LIN {X 0,Y 340.735,Z 431.04,A -85,B 0,C 180,E1 -14001.773,E2 -14001.773} C_VEL
LIN {X 0,Y 340.725,Z 431.04,A -85,B 0,C 180,E1 -14005.595,E2 -14005.595} C_VEL
LIN {X 0,Y 340.733,Z 431.068,A -85,B 0,C 180,E1 -14009.845,E2 -14009.845} C_VEL
LIN {X 0,Y 343.877,Z 445.891,A -85,B 0,C 180,E1 -14012.952,E2 -14012.952} C_VEL
LIN {X 0,Y 345.184,Z 453.139,A -85,B 0,C 180,E1 -14014.437,E2 -14014.437} C_VEL
LIN {X 0,Y 344.329,Z 467.534,A -85,B 0,C 180,E1 -14017.182,E2 -14017.182} C_VEL
LIN {X 0,Y 343.997,Z 473.692,A -85,B 0,C 180,E1 -14018.325,E2 -14018.325} C_VEL
LIN {X 0,Y 347.393,Z 500.288,A -85,B 0,C 180,E1 -14019.239,E2 -14019.239} C_VEL
LIN {X 0,Y 345.062,Z 584.431,A -85,B 0,C 180,E1 -14021.597,E2 -14021.597} C_VEL
LIN {X 0,Y 344.476,Z 598.904,A -85,B 0,C 180,E1 -14022.256,E2 -14022.256} C_VEL
LIN {X 0,Y 343.764,Z 611.4,A -85,B 0,C 180,E1 -14023.062,E2 -14023.062} C_VEL
LIN {X 0,Y 343.031,Z 623.647,A -85,B 0,C 180,E1 -14024.096,E2 -14024.096} C_VEL
LIN {X 0,Y 342.314,Z 634.938,A -85,B 0,C 180,E1 -14025.308,E2 -14025.308} C_VEL
LIN {X 0,Y 341.516,Z 645.889,A -85,B 0,C 180,E1 -14026.765,E2 -14026.765} C_VEL
LIN {X 0,Y 340.688,Z 655.695,A -85,B 0,C 180,E1 -14028.397,E2 -14028.397} C_VEL
LIN {X 0,Y 340.179,Z 663.039,A -85,B 0,C 180,E1 -14029.886,E2 -14029.886} C_VEL
LIN {X 0,Y 339.671,Z 670.234,A -85,B 0,C 180,E1 -14031.672,E2 -14031.672} C_VEL
LIN {X 0,Y 339.338,Z 676.847,A -85,B 0,C 180,E1 -14033.788,E2 -14033.788} C_VEL
LIN {X 0,Y 339.206,Z 681.571,A -85,B 0,C 180,E1 -14035.841,E2 -14035.841} C_VEL
LIN {X 0,Y 339.05,Z 684.475,A -85,B 0,C 180,E1 -14037.624,E2 -14037.624} C_VEL
LIN {X 0,Y 339.018,Z 685.837,A -85,B 0,C 180,E1 -14038.812,E2 -14038.812} C_VEL
LIN {X 0,Y 339.046,Z 686.75,A -85,B 0,C 180,E1 -14040,E2 -14040} C_VEL
LIN {X 0,Y 339.08,Z 687.194,A -85,B 0,C 180,E1 -14041.188,E2 -14041.188} C_VEL
LIN {X 0,Y 339.136,Z 687.227,A -85,B 0,C 180,E1 -14042.375,E2 -14042.375} C_VEL
LIN {X 0,Y 339.212,Z 686.82,A -85,B 0,C 180,E1 -14043.564,E2 -14043.564} C_VEL
LIN {X 0,Y 339.398,Z 685.947,A -85,B 0,C 180,E1 -14044.751,E2 -14044.751} C_VEL
LIN {X 0,Y 339.705,Z 684.655,A -85,B 0,C 180,E1 -14045.937,E2 -14045.937} C_VEL
LIN {X 0,Y 340.059,Z 681.86,A -85,B 0,C 180,E1 -14047.72,E2 -14047.72} C_VEL
LIN {X 0,Y 340.682,Z 677.987,A -85,B 0,C 180,E1 -14049.499,E2 -14049.499} C_VEL
LIN {X 0,Y 341.571,Z 672.921,A -85,B 0,C 180,E1 -14051.272,E2 -14051.272} C_VEL
LIN {X 0,Y 342.61,Z 666.526,A -85,B 0,C 180,E1 -14053.041,E2 -14053.041} C_VEL
LIN {X 0,Y 344.049,Z 658.543,A -85,B 0,C 180,E1 -14054.794,E2 -14054.794} C_VEL
LIN {X 0,Y 345.341,Z 650.417,A -85,B 0,C 180,E1 -14056.25,E2 -14056.25} C_VEL
LIN {X 0,Y 346.911,Z 640.605,A -85,B 0,C 180,E1 -14057.691,E2 -14057.691} C_VEL
LIN {X 0,Y 348.482,Z 629.771,A -85,B 0,C 180,E1 -14058.978,E2 -14058.978} C_VEL
LIN {X 0,Y 349.949,Z 617.73,A -85,B 0,C 180,E1 -14060.116,E2 -14060.116} C_VEL
LIN {X 0,Y 351.321,Z 605.219,A -85,B 0,C 180,E1 -14061.028,E2 -14061.028} C_VEL
LIN {X 0,Y 352.474,Z 591.942,A -85,B 0,C 180,E1 -14061.761,E2 -14061.761} C_VEL
LIN {X 0,Y 353.611,Z 575.675,A -85,B 0,C 180,E1 -14062.34,E2 -14062.34} C_VEL
LIN {X 0,Y 357.891,Z 509.779,A -85,B 0,C 180,E1 -14064.477,E2 -14064.477} C_VEL
LIN {X 0,Y 358.21,Z 503.514,A -85,B 0,C 180,E1 -14064.704,E2 -14064.704} C_VEL
LIN {X 0,Y 355.972,Z 490.842,A -85,B 0,C 180,E1 -14065.568,E2 -14065.568} C_VEL
LIN {X 0,Y 352.614,Z 476.312,A -85,B 0,C 180,E1 -14066.788,E2 -14066.788} C_VEL
LIN {X 0,Y 353.362,Z 470.45,A -85,B 0,C 180,E1 -14068.018,E2 -14068.018} C_VEL
LIN {X 0,Y 352.553,Z 464.536,A -85,B 0,C 180,E1 -14069.563,E2 -14069.563} C_VEL
LIN {X 0,Y 351.253,Z 458.463,A -85,B 0,C 180,E1 -14071.347,E2 -14071.347} C_VEL
LIN {X 0,Y 349.357,Z 451.655,A -85,B 0,C 180,E1 -14073.608,E2 -14073.608} C_VEL
LIN {X 0,Y 347.334,Z 445.631,A -85,B 0,C 180,E1 -14075.966,E2 -14075.966} C_VEL
LIN {X 0,Y 344.64,Z 439.216,A -85,B 0,C 180,E1 -14079.21,E2 -14079.21} C_VEL
LIN {X 0,Y 342.538,Z 434.998,A -85,B 0,C 180,E1 -14082.385,E2 -14082.385} C_VEL
LIN {X 0,Y 341.197,Z 433.028,A -85,B 0,C 180,E1 -14085.546,E2 -14085.546} C_VEL
LIN {X 0,Y 341.086,Z 432.671,A -85,B 0,C 180,E1 -14087.883,E2 -14087.883} C_VEL
LIN {X 0,Y 341.624,Z 433.725,A -85,B 0,C 180,E1 -14090.376,E2 -14090.376} C_VEL
LIN {X 0,Y 343.462,Z 435.825,A -85,B 0,C 180,E1 -14092.942,E2 -14092.942} C_VEL
LIN {X 0,Y 345.596,Z 439.87,A -85,B 0,C 180,E1 -14095.291,E2 -14095.291} C_VEL
LIN {X 0,Y 346.763,Z 441.759,A -85,B 0,C 180,E1 -14096.198,E2 -14096.198} C_VEL
LIN {X 0,Y 347.63,Z 443.646,A -85,B 0,C 180,E1 -14096.917,E2 -14096.917} C_VEL
LIN {X 0,Y 348.918,Z 451.136,A -85,B 0,C 180,E1 -14098.688,E2 -14098.688} C_VEL
LIN {X 0,Y 351.16,Z 461.414,A -85,B 0,C 180,E1 -14100.754,E2 -14100.754} C_VEL
LIN {X 0,Y 351.367,Z 473.128,A -85,B 0,C 180,E1 -14102.219,E2 -14102.219} C_VEL
LIN {X 0,Y 351.904,Z 484.135,A -85,B 0,C 180,E1 -14103.426,E2 -14103.426} C_VEL
LIN {X 0,Y 354.222,Z 500.627,A -85,B 0,C 180,E1 -14104.573,E2 -14104.573} C_VEL
LIN {X 0,Y 355.496,Z 514.817,A -85,B 0,C 180,E1 -14105.395,E2 -14105.395} C_VEL
LIN {X 0,Y 355.953,Z 529.982,A -85,B 0,C 180,E1 -14106.106,E2 -14106.106} C_VEL
LIN {X 0,Y 351.819,Z 594.042,A -85,B 0,C 180,E1 -14108.234,E2 -14108.234} C_VEL
LIN {X 0,Y 350.644,Z 610.198,A -85,B 0,C 180,E1 -14108.814,E2 -14108.814} C_VEL
LIN {X 0,Y 349.293,Z 624.619,A -85,B 0,C 180,E1 -14109.614,E2 -14109.614} C_VEL
LIN {X 0,Y 347.641,Z 638.466,A -85,B 0,C 180,E1 -14110.668,E2 -14110.668} C_VEL
LIN {X 0,Y 346.154,Z 649.931,A -85,B 0,C 180,E1 -14111.81,E2 -14111.81} C_VEL
LIN {X 0,Y 344.724,Z 660.329,A -85,B 0,C 180,E1 -14113.111,E2 -14113.111} C_VEL
LIN {X 0,Y 343.335,Z 669.83,A -85,B 0,C 180,E1 -14114.567,E2 -14114.567} C_VEL
LIN {X 0,Y 342.004,Z 679.094,A -85,B 0,C 180,E1 -14116.331,E2 -14116.331} C_VEL
LIN {X 0,Y 340.926,Z 686.559,A -85,B 0,C 180,E1 -14118.103,E2 -14118.103} C_VEL
LIN {X 0,Y 340.164,Z 692.472,A -85,B 0,C 180,E1 -14119.885,E2 -14119.885} C_VEL
LIN {X 0,Y 339.571,Z 697.133,A -85,B 0,C 180,E1 -14121.67,E2 -14121.67} C_VEL
LIN {X 0,Y 339.376,Z 699.6,A -85,B 0,C 180,E1 -14122.862,E2 -14122.862} C_VEL
LIN {X 0,Y 339.21,Z 701.57,A -85,B 0,C 180,E1 -14124.054,E2 -14124.054} C_VEL
LIN {X 0,Y 339.155,Z 703.047,A -85,B 0,C 180,E1 -14125.245,E2 -14125.245} C_VEL
LIN {X 0,Y 339.129,Z 704.098,A -85,B 0,C 180,E1 -14126.436,E2 -14126.436} C_VEL
LIN {X 0,Y 339.056,Z 704.68,A -85,B 0,C 180,E1 -14127.624,E2 -14127.624} C_VEL
LIN {X 0,Y 339.14,Z 705.07,A -85,B 0,C 180,E1 -14130,E2 -14130} C_VEL
LIN {X 0,Y 339.076,Z 704.844,A -85,B 0,C 180,E1 -14131.188,E2 -14131.188} C_VEL
LIN {X 0,Y 339.128,Z 703.216,A -85,B 0,C 180,E1 -14133.564,E2 -14133.564} C_VEL
LIN {X 0,Y 339.137,Z 701.78,A -85,B 0,C 180,E1 -14134.755,E2 -14134.755} C_VEL
LIN {X 0,Y 339.239,Z 698.795,A -85,B 0,C 180,E1 -14136.543,E2 -14136.543} C_VEL
LIN {X 0,Y 339.533,Z 694.746,A -85,B 0,C 180,E1 -14138.331,E2 -14138.331} C_VEL
LIN {X 0,Y 340.098,Z 688.503,A -85,B 0,C 180,E1 -14140.417,E2 -14140.417} C_VEL
LIN {X 0,Y 340.817,Z 681.692,A -85,B 0,C 180,E1 -14142.202,E2 -14142.202} C_VEL
LIN {X 0,Y 341.715,Z 674.725,A -85,B 0,C 180,E1 -14143.681,E2 -14143.681} C_VEL
LIN {X 0,Y 342.727,Z 666.304,A -85,B 0,C 180,E1 -14145.156,E2 -14145.156} C_VEL
LIN {X 0,Y 343.843,Z 655.879,A -85,B 0,C 180,E1 -14146.628,E2 -14146.628} C_VEL
LIN {X 0,Y 345.026,Z 645.554,A -85,B 0,C 180,E1 -14147.791,E2 -14147.791} C_VEL
LIN {X 0,Y 346.817,Z 629.693,A -85,B 0,C 180,E1 -14149.226,E2 -14149.226} C_VEL
LIN {X 0,Y 348.632,Z 617.052,A -85,B 0,C 180,E1 -14150.349,E2 -14150.349} C_VEL
LIN {X 0,Y 350.406,Z 603.79,A -85,B 0,C 180,E1 -14151.24,E2 -14151.24} C_VEL
LIN {X 0,Y 351.896,Z 589.543,A -85,B 0,C 180,E1 -14151.953,E2 -14151.953} C_VEL
LIN {X 0,Y 353.266,Z 568.128,A -85,B 0,C 180,E1 -14152.672,E2 -14152.672} C_VEL
LIN {X 0,Y 355.655,Z 527.031,A -85,B 0,C 180,E1 -14154.004,E2 -14154.004} C_VEL
LIN {X 0,Y 354.885,Z 512.697,A -85,B 0,C 180,E1 -14154.691,E2 -14154.691} C_VEL
LIN {X 0,Y 353.058,Z 496.809,A -85,B 0,C 180,E1 -14155.62,E2 -14155.62} C_VEL
LIN {X 0,Y 350.219,Z 481.179,A -85,B 0,C 180,E1 -14156.748,E2 -14156.748} C_VEL
LIN {X 0,Y 347.992,Z 470.293,A -85,B 0,C 180,E1 -14157.678,E2 -14157.678} C_VEL
LIN {X 0,Y 349.181,Z 463.767,A -85,B 0,C 180,E1 -14159.276,E2 -14159.276} C_VEL
LIN {X 0,Y 348.37,Z 458.198,A -85,B 0,C 180,E1 -14160.96,E2 -14160.96} C_VEL
LIN {X 0,Y 346.425,Z 449.389,A -85,B 0,C 180,E1 -14164.025,E2 -14164.025} C_VEL
LIN {X 0,Y 344.561,Z 442.807,A -85,B 0,C 180,E1 -14166.83,E2 -14166.83} C_VEL
LIN {X 0,Y 342.932,Z 437.851,A -85,B 0,C 180,E1 -14169.443,E2 -14169.443} C_VEL
LIN {X 0,Y 341.61,Z 433.699,A -85,B 0,C 180,E1 -14172.214,E2 -14172.214} C_VEL
LIN {X 0,Y 340.674,Z 431.049,A -85,B 0,C 180,E1 -14174.771,E2 -14174.771} C_VEL
LIN {X 0,Y 340.688,Z 431.048,A -85,B 0,C 180,E1 -14178.691,E2 -14178.691} C_VEL
LIN {X 0,Y 340.735,Z 431.041,A -85,B 0,C 180,E1 -14181.773,E2 -14181.773} C_VEL
LIN {X 0,Y 340.725,Z 431.041,A -85,B 0,C 180,E1 -14185.595,E2 -14185.595} C_VEL
LIN {X 0,Y 340.712,Z 431.274,A -85,B 0,C 180,E1 -14187.75,E2 -14187.75} C_VEL
LIN {X 0,Y 341.859,Z 434.768,A -85,B 0,C 180,E1 -14191.111,E2 -14191.111} C_VEL
LIN {X 0,Y 342.024,Z 435.219,A -85,B 0,C 180,E1 -14191.378,E2 -14191.378} C_VEL
LIN {X 0,Y 344.364,Z 438.406,A -85,B 0,C 180,E1 -14192.051,E2 -14192.051} C_VEL
LIN {X 0,Y 346.208,Z 440.911,A -85,B 0,C 180,E1 -14192.546,E2 -14192.546} C_VEL
LIN {X 0,Y 348.676,Z 444.26,A -85,B 0,C 180,E1 -14193.177,E2 -14193.177} C_VEL
LIN {X 0,Y 352.353,Z 449.838,A -85,B 0,C 180,E1 -14194.091,E2 -14194.091} C_VEL
LIN {X 0,Y 357.826,Z 460.119,A -85,B 0,C 180,E1 -14195.413,E2 -14195.413} C_VEL
LIN {X 0,Y 358.798,Z 462.095,A -85,B 0,C 180,E1 -14195.634,E2 -14195.634} C_VEL
LIN {X 0,Y 354.278,Z 529.936,A -85,B 0,C 180,E1 -14197.896,E2 -14197.896} C_VEL
LIN {X 0,Y 353.504,Z 543.651,A -85,B 0,C 180,E1 -14198.497,E2 -14198.497} C_VEL
LIN {X 0,Y 352.576,Z 556.471,A -85,B 0,C 180,E1 -14199.31,E2 -14199.31} C_VEL
LIN {X 0,Y 351.311,Z 568.751,A -85,B 0,C 180,E1 -14200.325,E2 -14200.325} C_VEL
LIN {X 0,Y 349.788,Z 580.474,A -85,B 0,C 180,E1 -14201.551,E2 -14201.551} C_VEL
LIN {X 0,Y 348.228,Z 591.315,A -85,B 0,C 180,E1 -14202.984,E2 -14202.984} C_VEL
LIN {X 0,Y 346.834,Z 600.035,A -85,B 0,C 180,E1 -14204.426,E2 -14204.426} C_VEL
LIN {X 0,Y 345.346,Z 608.53,A -85,B 0,C 180,E1 -14206.165,E2 -14206.165} C_VEL
LIN {X 0,Y 344.008,Z 615.427,A -85,B 0,C 180,E1 -14207.913,E2 -14207.913} C_VEL
LIN {X 0,Y 342.812,Z 621.479,A -85,B 0,C 180,E1 -14209.92,E2 -14209.92} C_VEL
LIN {X 0,Y 341.723,Z 625.627,A -85,B 0,C 180,E1 -14211.723,E2 -14211.723} C_VEL
LIN {X 0,Y 341.324,Z 627.682,A -85,B 0,C 180,E1 -14212.903,E2 -14212.903} C_VEL
LIN {X 0,Y 340.956,Z 629.248,A -85,B 0,C 180,E1 -14214.084,E2 -14214.084} C_VEL
LIN {X 0,Y 340.574,Z 630.401,A -85,B 0,C 180,E1 -14215.265,E2 -14215.265} C_VEL
LIN {X 0,Y 340.191,Z 631.145,A -85,B 0,C 180,E1 -14216.447,E2 -14216.447} C_VEL
LIN {X 0,Y 339.906,Z 631.432,A -85,B 0,C 180,E1 -14217.63,E2 -14217.63} C_VEL
LIN {X 0,Y 339.749,Z 631.264,A -85,B 0,C 180,E1 -14218.815,E2 -14218.815} C_VEL
LIN {X 0,Y 339.693,Z 630.677,A -85,B 0,C 180,E1 -14220,E2 -14220} C_VEL
LIN {X 0,Y 339.712,Z 629.667,A -85,B 0,C 180,E1 -14221.185,E2 -14221.185} C_VEL
LIN {X 0,Y 339.747,Z 628.188,A -85,B 0,C 180,E1 -14222.371,E2 -14222.371} C_VEL
LIN {X 0,Y 340,Z 625.148,A -85,B 0,C 180,E1 -14224.149,E2 -14224.149} C_VEL
LIN {X 0,Y 340.097,Z 621.032,A -85,B 0,C 180,E1 -14225.931,E2 -14225.931} C_VEL
LIN {X 0,Y 340.449,Z 614.758,A -85,B 0,C 180,E1 -14227.993,E2 -14227.993} C_VEL
LIN {X 0,Y 340.865,Z 607.712,A -85,B 0,C 180,E1 -14229.794,E2 -14229.794} C_VEL
LIN {X 0,Y 341.507,Z 599.031,A -85,B 0,C 180,E1 -14231.575,E2 -14231.575} C_VEL
LIN {X 0,Y 342.216,Z 589.175,A -85,B 0,C 180,E1 -14233.207,E2 -14233.207} C_VEL
LIN {X 0,Y 342.969,Z 578.054,A -85,B 0,C 180,E1 -14234.69,E2 -14234.69} C_VEL
LIN {X 0,Y 343.696,Z 566.966,A -85,B 0,C 180,E1 -14235.88,E2 -14235.88} C_VEL
LIN {X 0,Y 344.25,Z 554.855,A -85,B 0,C 180,E1 -14236.913,E2 -14236.913} C_VEL
LIN {X 0,Y 344.841,Z 542.538,A -85,B 0,C 180,E1 -14237.724,E2 -14237.724} C_VEL
LIN {X 0,Y 345.26,Z 529.261,A -85,B 0,C 180,E1 -14238.354,E2 -14238.354} C_VEL
LIN {X 0,Y 345.75,Z 507.069,A -85,B 0,C 180,E1 -14239.017,E2 -14239.017} C_VEL
LIN {X 0,Y 347.211,Z 450.909,A -85,B 0,C 180,E1 -14240.587,E2 -14240.587} C_VEL
LIN {X 0,Y 340.756,Z 431.041,A -85,B 0,C 180,E1 -14241.464,E2 -14241.464} C_VEL
LIN {X 0,Y 340.774,Z 431.037,A -85,B 0,C 180,E1 -14245.664,E2 -14245.664} C_VEL
LIN {X 0,Y 340.731,Z 431.036,A -85,B 0,C 180,E1 -14248.321,E2 -14248.321} C_VEL
LIN {X 0,Y 340.7,Z 431.043,A -85,B 0,C 180,E1 -14251.045,E2 -14251.045} C_VEL
LIN {X 0,Y 340.72,Z 431.031,A -85,B 0,C 180,E1 -14255.279,E2 -14255.279} C_VEL
LIN {X 0,Y 340.712,Z 431.046,A -85,B 0,C 180,E1 -14258.386,E2 -14258.386} C_VEL
LIN {X 0,Y 340.701,Z 431.043,A -85,B 0,C 180,E1 -14262.045,E2 -14262.045} C_VEL
LIN {X 0,Y 340.654,Z 431.038,A -85,B 0,C 180,E1 -14266.227,E2 -14266.227} C_VEL
LIN {X 0,Y 340.69,Z 431.038,A -85,B 0,C 180,E1 -14269.753,E2 -14269.753} C_VEL
LIN {X 0,Y 340.707,Z 431.039,A -85,B 0,C 180,E1 -14273.258,E2 -14273.258} C_VEL
LIN {X 0,Y 340.694,Z 431.043,A -85,B 0,C 180,E1 -14276.153,E2 -14276.153} C_VEL
LIN {X 0,Y 340.73,Z 431.151,A -85,B 0,C 180,E1 -14278.076,E2 -14278.076} C_VEL
LIN {X 0,Y 343.807,Z 443.339,A -85,B 0,C 180,E1 -14280.861,E2 -14280.861} C_VEL
LIN {X 0,Y 346.36,Z 455.442,A -85,B 0,C 180,E1 -14283.487,E2 -14283.487} C_VEL
LIN {X 0,Y 346.577,Z 458.765,A -85,B 0,C 180,E1 -14284.152,E2 -14284.152} C_VEL
LIN {X 0,Y 345.729,Z 472.884,A -85,B 0,C 180,E1 -14286.703,E2 -14286.703} C_VEL
LIN {X 0,Y 350.593,Z 500.147,A -85,B 0,C 180,E1 -14287.657,E2 -14287.657} C_VEL
LIN {X 0,Y 349.247,Z 578.094,A -85,B 0,C 180,E1 -14289.265,E2 -14289.265} C_VEL
LIN {X 0,Y 348.779,Z 591.322,A -85,B 0,C 180,E1 -14289.66,E2 -14289.66} C_VEL
LIN {X 0,Y 347.957,Z 604.505,A -85,B 0,C 180,E1 -14290.303,E2 -14290.303} C_VEL
LIN {X 0,Y 347.044,Z 616.117,A -85,B 0,C 180,E1 -14291.094,E2 -14291.094} C_VEL
LIN {X 0,Y 346.027,Z 627.47,A -85,B 0,C 180,E1 -14292.11,E2 -14292.11} C_VEL
LIN {X 0,Y 344.956,Z 637.518,A -85,B 0,C 180,E1 -14293.249,E2 -14293.249} C_VEL
LIN {X 0,Y 343.897,Z 647.105,A -85,B 0,C 180,E1 -14294.593,E2 -14294.593} C_VEL
LIN {X 0,Y 342.683,Z 655.692,A -85,B 0,C 180,E1 -14296.056,E2 -14296.056} C_VEL
LIN {X 0,Y 341.809,Z 662.776,A -85,B 0,C 180,E1 -14297.532,E2 -14297.532} C_VEL
LIN {X 0,Y 340.928,Z 669.734,A -85,B 0,C 180,E1 -14299.308,E2 -14299.308} C_VEL
LIN {X 0,Y 340.14,Z 675.264,A -85,B 0,C 180,E1 -14301.085,E2 -14301.085} C_VEL
LIN {X 0,Y 339.728,Z 679.599,A -85,B 0,C 180,E1 -14302.87,E2 -14302.87} C_VEL
LIN {X 0,Y 339.498,Z 681.88,A -85,B 0,C 180,E1 -14304.059,E2 -14304.059} C_VEL
LIN {X 0,Y 339.344,Z 683.74,A -85,B 0,C 180,E1 -14305.248,E2 -14305.248} C_VEL
LIN {X 0,Y 339.176,Z 685.162,A -85,B 0,C 180,E1 -14306.436,E2 -14306.436} C_VEL
LIN {X 0,Y 339.057,Z 686.771,A -85,B 0,C 180,E1 -14308.812,E2 -14308.812} C_VEL
LIN {X 0,Y 339.054,Z 687.005,A -85,B 0,C 180,E1 -14310,E2 -14310} C_VEL
LIN {X 0,Y 339.057,Z 686.812,A -85,B 0,C 180,E1 -14311.188,E2 -14311.188} C_VEL
LIN {X 0,Y 339.176,Z 685.257,A -85,B 0,C 180,E1 -14313.564,E2 -14313.564} C_VEL
LIN {X 0,Y 339.341,Z 683.889,A -85,B 0,C 180,E1 -14314.752,E2 -14314.752} C_VEL
LIN {X 0,Y 339.614,Z 680.838,A -85,B 0,C 180,E1 -14316.626,E2 -14316.626} C_VEL
LIN {X 0,Y 339.979,Z 677.11,A -85,B 0,C 180,E1 -14318.32,E2 -14318.32} C_VEL
LIN {X 0,Y 340.594,Z 672.047,A -85,B 0,C 180,E1 -14320.102,E2 -14320.102} C_VEL
LIN {X 0,Y 341.433,Z 665.663,A -85,B 0,C 180,E1 -14321.879,E2 -14321.879} C_VEL
LIN {X 0,Y 342.446,Z 657.73,A -85,B 0,C 180,E1 -14323.651,E2 -14323.651} C_VEL
LIN {X 0,Y 343.587,Z 649.617,A -85,B 0,C 180,E1 -14325.118,E2 -14325.118} C_VEL
LIN {X 0,Y 344.745,Z 639.639,A -85,B 0,C 180,E1 -14326.583,E2 -14326.583} C_VEL
LIN {X 0,Y 345.852,Z 629.069,A -85,B 0,C 180,E1 -14327.828,E2 -14327.828} C_VEL
LIN {X 0,Y 345.787,Z 624.105,A -85,B 0,C 180,E1 -14328.359,E2 -14328.359} C_VEL
LIN {X 0,Y 343.871,Z 615.904,A -85,B 0,C 180,E1 -14329.229,E2 -14329.229} C_VEL
LIN {X 0,Y 341.847,Z 607.372,A -85,B 0,C 180,E1 -14329.998,E2 -14329.998} C_VEL
LIN {X 0,Y 341.6,Z 601.893,A -85,B 0,C 180,E1 -14330.361,E2 -14330.361} C_VEL
LIN {X 0,Y 342.202,Z 589.178,A -85,B 0,C 180,E1 -14330.946,E2 -14330.946} C_VEL
LIN {X 0,Y 342.727,Z 575.953,A -85,B 0,C 180,E1 -14331.306,E2 -14331.306} C_VEL
LIN {X 0,Y 344.073,Z 501.274,A -85,B 0,C 180,E1 -14332.874,E2 -14332.874} C_VEL
LIN {X 0,Y 339.44,Z 475.293,A -85,B 0,C 180,E1 -14333.795,E2 -14333.795} C_VEL
LIN {X 0,Y 339.048,Z 472.783,A -85,B 0,C 180,E1 -14333.933,E2 -14333.933} C_VEL
LIN {X 0,Y 339.88,Z 459.482,A -85,B 0,C 180,E1 -14336.381,E2 -14336.381} C_VEL
LIN {X 0,Y 338.309,Z 450.963,A -85,B 0,C 180,E1 -14338.204,E2 -14338.204} C_VEL
LIN {X 0,Y 335.381,Z 438.328,A -85,B 0,C 180,E1 -14341.086,E2 -14341.086} C_VEL
LIN {X 0,Y 333.648,Z 431.927,A -85,B 0,C 180,E1 -14342.588,E2 -14342.588} C_VEL
LIN {X 0,Y 333.678,Z 431.925,A -85,B 0,C 180,E1 -14346.139,E2 -14346.139} C_VEL
LIN {X 0,Y 333.649,Z 431.924,A -85,B 0,C 180,E1 -14349.192,E2 -14349.192} C_VEL
LIN {X 0,Y 333.635,Z 431.928,A -85,B 0,C 180,E1 -14352.5,E2 -14352.5} C_VEL
LIN {X 0,Y 333.625,Z 431.93,A -85,B 0,C 180,E1 -14355.959,E2 -14355.959} C_VEL
LIN {X 0,Y 333.649,Z 431.92,A -85,B 0,C 180,E1 -14359.315,E2 -14359.315} C_VEL
LIN {X 0,Y 333.667,Z 431.905,A -85,B 0,C 180,E1 -14363.168,E2 -14363.168} C_VEL
LIN {X 0,Y 333.676,Z 431.919,A -85,B 0,C 180,E1 -14365.341,E2 -14365.341} C_VEL
LIN {X 0,Y 333.694,Z 432.008,A -85,B 0,C 180,E1 -14369.594,E2 -14369.594} C_VEL
LIN {X 0,Y 337.063,Z 447.88,A -85,B 0,C 180,E1 -14372.964,E2 -14372.964} C_VEL
LIN {X 0,Y 338.139,Z 453.443,A -85,B 0,C 180,E1 -14374.121,E2 -14374.121} C_VEL
LIN {X 0,Y 337.619,Z 464.884,A -85,B 0,C 180,E1 -14376.337,E2 -14376.337} C_VEL
LIN {X 0,Y 337.043,Z 473.676,A -85,B 0,C 180,E1 -14378.029,E2 -14378.029} C_VEL
LIN {X 0,Y 340.484,Z 500.87,A -85,B 0,C 180,E1 -14378.997,E2 -14378.997} C_VEL
LIN {X 0,Y 338.043,Z 585.238,A -85,B 0,C 180,E1 -14381.437,E2 -14381.437} C_VEL
LIN {X 0,Y 337.444,Z 599.489,A -85,B 0,C 180,E1 -14382.109,E2 -14382.109} C_VEL
LIN {X 0,Y 336.634,Z 612.818,A -85,B 0,C 180,E1 -14383.005,E2 -14383.005} C_VEL
LIN {X 0,Y 335.894,Z 624.819,A -85,B 0,C 180,E1 -14384.061,E2 -14384.061} C_VEL
LIN {X 0,Y 335.164,Z 636.935,A -85,B 0,C 180,E1 -14385.426,E2 -14385.426} C_VEL
LIN {X 0,Y 334.485,Z 645.726,A -85,B 0,C 180,E1 -14386.637,E2 -14386.637} C_VEL
LIN {X 0,Y 333.691,Z 654.815,A -85,B 0,C 180,E1 -14388.15,E2 -14388.15} C_VEL
LIN {X 0,Y 333.039,Z 663.705,A -85,B 0,C 180,E1 -14389.974,E2 -14389.974} C_VEL
LIN {X 0,Y 332.563,Z 670.799,A -85,B 0,C 180,E1 -14391.799,E2 -14391.799} C_VEL
LIN {X 0,Y 332.221,Z 677.252,A -85,B 0,C 180,E1 -14393.928,E2 -14393.928} C_VEL
LIN {X 0,Y 332.122,Z 681.407,A -85,B 0,C 180,E1 -14395.753,E2 -14395.753} C_VEL
LIN {X 0,Y 331.967,Z 684.423,A -85,B 0,C 180,E1 -14397.573,E2 -14397.573} C_VEL
LIN {X 0,Y 331.924,Z 685.841,A -85,B 0,C 180,E1 -14398.787,E2 -14398.787} C_VEL
LIN {X 0,Y 331.949,Z 686.845,A -85,B 0,C 180,E1 -14400,E2 -14400} C_VEL
LIN {X 0,Y 331.985,Z 687.375,A -85,B 0,C 180,E1 -14401.213,E2 -14401.213} C_VEL
LIN {X 0,Y 332.049,Z 687.466,A -85,B 0,C 180,E1 -14402.426,E2 -14402.426} C_VEL
LIN {X 0,Y 332.142,Z 687.143,A -85,B 0,C 180,E1 -14403.639,E2 -14403.639} C_VEL
LIN {X 0,Y 332.351,Z 686.343,A -85,B 0,C 180,E1 -14404.852,E2 -14404.852} C_VEL
LIN {X 0,Y 332.798,Z 683.878,A -85,B 0,C 180,E1 -14407,E2 -14407} C_VEL
LIN {X 0,Y 333.468,Z 680.103,A -85,B 0,C 180,E1 -14409.095,E2 -14409.095} C_VEL
LIN {X 0,Y 334.351,Z 675.57,A -85,B 0,C 180,E1 -14410.905,E2 -14410.905} C_VEL
LIN {X 0,Y 335.557,Z 668.694,A -85,B 0,C 180,E1 -14413.012,E2 -14413.012} C_VEL
LIN {X 0,Y 337.007,Z 661.231,A -85,B 0,C 180,E1 -14414.801,E2 -14414.801} C_VEL
LIN {X 0,Y 338.369,Z 653.636,A -85,B 0,C 180,E1 -14416.284,E2 -14416.284} C_VEL
LIN {X 0,Y 340.028,Z 644.063,A -85,B 0,C 180,E1 -14417.813,E2 -14417.813} C_VEL
LIN {X 0,Y 341.741,Z 633.196,A -85,B 0,C 180,E1 -14419.211,E2 -14419.211} C_VEL
LIN {X 0,Y 343.333,Z 622.142,A -85,B 0,C 180,E1 -14420.364,E2 -14420.364} C_VEL
LIN {X 0,Y 344.862,Z 609.89,A -85,B 0,C 180,E1 -14421.363,E2 -14421.363} C_VEL
LIN {X 0,Y 346.124,Z 597.493,A -85,B 0,C 180,E1 -14422.142,E2 -14422.142} C_VEL
LIN {X 0,Y 347.316,Z 583.091,A -85,B 0,C 180,E1 -14422.768,E2 -14422.768} C_VEL
LIN {X 0,Y 352.794,Z 505.642,A -85,B 0,C 180,E1 -14425.363,E2 -14425.363} C_VEL
LIN {X 0,Y 350.797,Z 493.497,A -85,B 0,C 180,E1 -14426.234,E2 -14426.234} C_VEL
LIN {X 0,Y 347.674,Z 479.394,A -85,B 0,C 180,E1 -14427.463,E2 -14427.463} C_VEL
LIN {X 0,Y 347.038,Z 476.536,A -85,B 0,C 180,E1 -14427.761,E2 -14427.761} C_VEL
LIN {X 0,Y 347.394,Z 472.968,A -85,B 0,C 180,E1 -14428.548,E2 -14428.548} C_VEL
LIN {X 0,Y 346.216,Z 465.172,A -85,B 0,C 180,E1 -14430.748,E2 -14430.748} C_VEL
LIN {X 0,Y 344.233,Z 457.04,A -85,B 0,C 180,E1 -14433.452,E2 -14433.452} C_VEL
LIN {X 0,Y 342.337,Z 450.942,A -85,B 0,C 180,E1 -14435.884,E2 -14435.884} C_VEL
LIN {X 0,Y 340.436,Z 446.072,A -85,B 0,C 180,E1 -14438.327,E2 -14438.327} C_VEL
LIN {X 0,Y 339.288,Z 443.511,A -85,B 0,C 180,E1 -14439.966,E2 -14439.966} C_VEL
LIN {X 0,Y 338.334,Z 441.303,A -85,B 0,C 180,E1 -14441.661,E2 -14441.661} C_VEL
LIN {X 0,Y 337.451,Z 439.778,A -85,B 0,C 180,E1 -14443.416,E2 -14443.416} C_VEL
LIN {X 0,Y 336.859,Z 438.418,A -85,B 0,C 180,E1 -14446.489,E2 -14446.489} C_VEL
LIN {X 0,Y 337.036,Z 438.632,A -85,B 0,C 180,E1 -14448.65,E2 -14448.65} C_VEL
LIN {X 0,Y 338.159,Z 440.394,A -85,B 0,C 180,E1 -14451.428,E2 -14451.428} C_VEL
LIN {X 0,Y 339.584,Z 442.118,A -85,B 0,C 180,E1 -14453.117,E2 -14453.117} C_VEL
LIN {X 0,Y 342.511,Z 447.257,A -85,B 0,C 180,E1 -14455.942,E2 -14455.942} C_VEL
LIN {X 0,Y 343.44,Z 449.705,A -85,B 0,C 180,E1 -14456.815,E2 -14456.815} C_VEL
LIN {X 0,Y 345.163,Z 460.513,A -85,B 0,C 180,E1 -14459.26,E2 -14459.26} C_VEL
LIN {X 0,Y 346.099,Z 464.668,A -85,B 0,C 180,E1 -14460.087,E2 -14460.087} C_VEL
LIN {X 0,Y 346.221,Z 475.224,A -85,B 0,C 180,E1 -14461.486,E2 -14461.486} C_VEL
LIN {X 0,Y 346.444,Z 483.85,A -85,B 0,C 180,E1 -14462.483,E2 -14462.483} C_VEL
LIN {X 0,Y 348.557,Z 498.928,A -85,B 0,C 180,E1 -14463.618,E2 -14463.618} C_VEL
LIN {X 0,Y 350.054,Z 514.876,A -85,B 0,C 180,E1 -14464.617,E2 -14464.617} C_VEL
LIN {X 0,Y 350.418,Z 530.269,A -85,B 0,C 180,E1 -14465.386,E2 -14465.386} C_VEL
LIN {X 0,Y 344.918,Z 607.297,A -85,B 0,C 180,E1 -14468.052,E2 -14468.052} C_VEL
LIN {X 0,Y 343.681,Z 620.288,A -85,B 0,C 180,E1 -14468.717,E2 -14468.717} C_VEL
LIN {X 0,Y 342.249,Z 632.431,A -85,B 0,C 180,E1 -14469.568,E2 -14469.568} C_VEL
LIN {X 0,Y 340.72,Z 643.64,A -85,B 0,C 180,E1 -14470.573,E2 -14470.573} C_VEL
LIN {X 0,Y 339.037,Z 655.101,A -85,B 0,C 180,E1 -14471.884,E2 -14471.884} C_VEL
LIN {X 0,Y 337.582,Z 664.921,A -85,B 0,C 180,E1 -14473.267,E2 -14473.267} C_VEL
LIN {X 0,Y 336.046,Z 674.042,A -85,B 0,C 180,E1 -14474.845,E2 -14474.845} C_VEL
LIN {X 0,Y 334.686,Z 682.385,A -85,B 0,C 180,E1 -14476.645,E2 -14476.645} C_VEL
LIN {X 0,Y 333.669,Z 689.148,A -85,B 0,C 180,E1 -14478.457,E2 -14478.457} C_VEL
LIN {X 0,Y 332.939,Z 694.48,A -85,B 0,C 180,E1 -14480.278,E2 -14480.278} C_VEL
LIN {X 0,Y 332.407,Z 698.594,A -85,B 0,C 180,E1 -14482.101,E2 -14482.101} C_VEL
LIN {X 0,Y 332.12,Z 701.729,A -85,B 0,C 180,E1 -14484.027,E2 -14484.027} C_VEL
LIN {X 0,Y 332.059,Z 703.026,A -85,B 0,C 180,E1 -14485.144,E2 -14485.144} C_VEL
LIN {X 0,Y 332.053,Z 704.01,A -85,B 0,C 180,E1 -14486.359,E2 -14486.359} C_VEL
LIN {X 0,Y 331.991,Z 704.67,A -85,B 0,C 180,E1 -14488.787,E2 -14488.787} C_VEL
LIN {X 0,Y 332.042,Z 704.881,A -85,B 0,C 180,E1 -14490,E2 -14490} C_VEL
LIN {X 0,Y 331.979,Z 704.655,A -85,B 0,C 180,E1 -14491.213,E2 -14491.213} C_VEL
LIN {X 0,Y 332.051,Z 703.027,A -85,B 0,C 180,E1 -14493.641,E2 -14493.641} C_VEL
LIN {X 0,Y 332.076,Z 699.997,A -85,B 0,C 180,E1 -14495.9,E2 -14495.9} C_VEL
LIN {X 0,Y 332.365,Z 696.009,A -85,B 0,C 180,E1 -14497.9,E2 -14497.9} C_VEL
LIN {X 0,Y 332.788,Z 691.191,A -85,B 0,C 180,E1 -14499.727,E2 -14499.727} C_VEL
LIN {X 0,Y 333.402,Z 685.094,A -85,B 0,C 180,E1 -14501.552,E2 -14501.552} C_VEL
LIN {X 0,Y 334.409,Z 677.497,A -85,B 0,C 180,E1 -14503.366,E2 -14503.366} C_VEL
LIN {X 0,Y 335.584,Z 668.106,A -85,B 0,C 180,E1 -14505.141,E2 -14505.141} C_VEL
LIN {X 0,Y 336.719,Z 658.216,A -85,B 0,C 180,E1 -14506.647,E2 -14506.647} C_VEL
LIN {X 0,Y 337.916,Z 648.2,A -85,B 0,C 180,E1 -14507.865,E2 -14507.865} C_VEL
LIN {X 0,Y 339.495,Z 634.856,A -85,B 0,C 180,E1 -14509.186,E2 -14509.186} C_VEL
LIN {X 0,Y 341.59,Z 622.078,A -85,B 0,C 180,E1 -14510.473,E2 -14510.473} C_VEL
LIN {X 0,Y 343.197,Z 611.58,A -85,B 0,C 180,E1 -14511.314,E2 -14511.314} C_VEL
LIN {X 0,Y 344.907,Z 598.324,A -85,B 0,C 180,E1 -14512.146,E2 -14512.146} C_VEL
LIN {X 0,Y 346.36,Z 584.169,A -85,B 0,C 180,E1 -14512.795,E2 -14512.795} C_VEL
LIN {X 0,Y 349.945,Z 527.866,A -85,B 0,C 180,E1 -14514.679,E2 -14514.679} C_VEL
LIN {X 0,Y 349.302,Z 514.056,A -85,B 0,C 180,E1 -14515.369,E2 -14515.369} C_VEL
LIN {X 0,Y 347.643,Z 498.628,A -85,B 0,C 180,E1 -14516.313,E2 -14516.313} C_VEL
LIN {X 0,Y 344.996,Z 483.241,A -85,B 0,C 180,E1 -14517.477,E2 -14517.477} C_VEL
LIN {X 0,Y 342.462,Z 471.523,A -85,B 0,C 180,E1 -14518.524,E2 -14518.524} C_VEL
LIN {X 0,Y 342.078,Z 468.976,A -85,B 0,C 180,E1 -14518.776,E2 -14518.776} C_VEL
LIN {X 0,Y 342.589,Z 466.145,A -85,B 0,C 180,E1 -14519.495,E2 -14519.495} C_VEL
LIN {X 0,Y 341.825,Z 460.54,A -85,B 0,C 180,E1 -14521.25,E2 -14521.25} C_VEL
LIN {X 0,Y 340.044,Z 452.324,A -85,B 0,C 180,E1 -14524.237,E2 -14524.237} C_VEL
LIN {X 0,Y 338.776,Z 447.432,A -85,B 0,C 180,E1 -14526.331,E2 -14526.331} C_VEL
LIN {X 0,Y 336.867,Z 441.494,A -85,B 0,C 180,E1 -14529.473,E2 -14529.473} C_VEL
LIN {X 0,Y 335.625,Z 437.668,A -85,B 0,C 180,E1 -14532.074,E2 -14532.074} C_VEL
LIN {X 0,Y 334.72,Z 435.126,A -85,B 0,C 180,E1 -14534.448,E2 -14534.448} C_VEL
LIN {X 0,Y 333.851,Z 432.972,A -85,B 0,C 180,E1 -14537.651,E2 -14537.651} C_VEL
LIN {X 0,Y 333.722,Z 432.341,A -85,B 0,C 180,E1 -14539.301,E2 -14539.301} C_VEL
LIN {X 0,Y 333.711,Z 432.21,A -85,B 0,C 180,E1 -14542.357,E2 -14542.357} C_VEL
LIN {X 0,Y 333.998,Z 433.297,A -85,B 0,C 180,E1 -14545.38,E2 -14545.38} C_VEL
LIN {X 0,Y 334.475,Z 434.408,A -85,B 0,C 180,E1 -14547.191,E2 -14547.191} C_VEL
LIN {X 0,Y 335.346,Z 437.025,A -85,B 0,C 180,E1 -14549.955,E2 -14549.955} C_VEL
LIN {X 0,Y 337.861,Z 440.383,A -85,B 0,C 180,E1 -14550.787,E2 -14550.787} C_VEL
LIN {X 0,Y 342.02,Z 445.734,A -85,B 0,C 180,E1 -14551.999,E2 -14551.999} C_VEL
LIN {X 0,Y 345.118,Z 450.159,A -85,B 0,C 180,E1 -14552.847,E2 -14552.847} C_VEL
LIN {X 0,Y 348.42,Z 455.366,A -85,B 0,C 180,E1 -14553.72,E2 -14553.72} C_VEL
LIN {X 0,Y 353.244,Z 464.773,A -85,B 0,C 180,E1 -14554.953,E2 -14554.953} C_VEL
LIN {X 0,Y 349.427,Z 515.747,A -85,B 0,C 180,E1 -14556.712,E2 -14556.712} C_VEL
LIN {X 0,Y 348.171,Z 537.01,A -85,B 0,C 180,E1 -14557.487,E2 -14557.487} C_VEL
LIN {X 0,Y 347.286,Z 549.756,A -85,B 0,C 180,E1 -14558.17,E2 -14558.17} C_VEL
LIN {X 0,Y 346.177,Z 562.042,A -85,B 0,C 180,E1 -14559.049,E2 -14559.049} C_VEL
LIN {X 0,Y 344.733,Z 573.959,A -85,B 0,C 180,E1 -14560.144,E2 -14560.144} C_VEL
LIN {X 0,Y 343.254,Z 584.327,A -85,B 0,C 180,E1 -14561.342,E2 -14561.342} C_VEL
LIN {X 0,Y 341.728,Z 593.517,A -85,B 0,C 180,E1 -14562.65,E2 -14562.65} C_VEL
LIN {X 0,Y 340.009,Z 603.567,A -85,B 0,C 180,E1 -14564.412,E2 -14564.412} C_VEL
LIN {X 0,Y 338.415,Z 611.534,A -85,B 0,C 180,E1 -14566.183,E2 -14566.183} C_VEL
LIN {X 0,Y 337.005,Z 617.916,A -85,B 0,C 180,E1 -14567.963,E2 -14567.963} C_VEL
LIN {X 0,Y 336.006,Z 622.616,A -85,B 0,C 180,E1 -14569.627,E2 -14569.627} C_VEL
LIN {X 0,Y 334.811,Z 626.859,A -85,B 0,C 180,E1 -14571.551,E2 -14571.551} C_VEL
LIN {X 0,Y 334.367,Z 628.813,A -85,B 0,C 180,E1 -14572.755,E2 -14572.755} C_VEL
LIN {X 0,Y 333.97,Z 630.296,A -85,B 0,C 180,E1 -14573.96,E2 -14573.96} C_VEL
LIN {X 0,Y 333.565,Z 631.371,A -85,B 0,C 180,E1 -14575.166,E2 -14575.166} C_VEL
LIN {X 0,Y 333.166,Z 632.023,A -85,B 0,C 180,E1 -14576.372,E2 -14576.372} C_VEL
LIN {X 0,Y 332.87,Z 632.205,A -85,B 0,C 180,E1 -14577.58,E2 -14577.58} C_VEL
LIN {X 0,Y 332.706,Z 631.971,A -85,B 0,C 180,E1 -14578.79,E2 -14578.79} C_VEL
LIN {X 0,Y 332.647,Z 631.319,A -85,B 0,C 180,E1 -14580,E2 -14580} C_VEL
LIN {X 0,Y 332.636,Z 630.2,A -85,B 0,C 180,E1 -14581.211,E2 -14581.211} C_VEL
LIN {X 0,Y 332.685,Z 628.647,A -85,B 0,C 180,E1 -14582.422,E2 -14582.422} C_VEL
LIN {X 0,Y 332.948,Z 625.469,A -85,B 0,C 180,E1 -14584.237,E2 -14584.237} C_VEL
LIN {X 0,Y 333.047,Z 621.203,A -85,B 0,C 180,E1 -14586.057,E2 -14586.057} C_VEL
LIN {X 0,Y 333.377,Z 615.044,A -85,B 0,C 180,E1 -14588.075,E2 -14588.075} C_VEL
LIN {X 0,Y 333.835,Z 607.5,A -85,B 0,C 180,E1 -14590.002,E2 -14590.002} C_VEL
LIN {X 0,Y 334.508,Z 598.636,A -85,B 0,C 180,E1 -14591.821,E2 -14591.821} C_VEL
LIN {X 0,Y 335.212,Z 588.486,A -85,B 0,C 180,E1 -14593.488,E2 -14593.488} C_VEL
LIN {X 0,Y 335.947,Z 578.325,A -85,B 0,C 180,E1 -14594.849,E2 -14594.849} C_VEL
LIN {X 0,Y 336.704,Z 567.061,A -85,B 0,C 180,E1 -14596.067,E2 -14596.067} C_VEL
LIN {X 0,Y 337.273,Z 554.869,A -85,B 0,C 180,E1 -14597.118,E2 -14597.118} C_VEL
LIN {X 0,Y 337.883,Z 542.352,A -85,B 0,C 180,E1 -14597.945,E2 -14597.945} C_VEL
LIN {X 0,Y 338.334,Z 527.739,A -85,B 0,C 180,E1 -14598.625,E2 -14598.625} C_VEL
LIN {X 0,Y 340.274,Z 452.148,A -85,B 0,C 180,E1 -14600.819,E2 -14600.819} C_VEL
LIN {X 0,Y 333.71,Z 431.916,A -85,B 0,C 180,E1 -14601.743,E2 -14601.743} C_VEL
LIN {X 0,Y 333.72,Z 431.915,A -85,B 0,C 180,E1 -14605.101,E2 -14605.101} C_VEL
LIN {X 0,Y 333.719,Z 431.908,A -85,B 0,C 180,E1 -14607.809,E2 -14607.809} C_VEL
LIN {X 0,Y 333.692,Z 431.918,A -85,B 0,C 180,E1 -14610.363,E2 -14610.363} C_VEL
LIN {X 0,Y 333.676,Z 431.901,A -85,B 0,C 180,E1 -14614.659,E2 -14614.659} C_VEL
LIN {X 0,Y 333.654,Z 431.925,A -85,B 0,C 180,E1 -14617.651,E2 -14617.651} C_VEL
LIN {X 0,Y 333.648,Z 431.908,A -85,B 0,C 180,E1 -14620.767,E2 -14620.767} C_VEL
LIN {X 0,Y 333.596,Z 431.932,A -85,B 0,C 180,E1 -14624.251,E2 -14624.251} C_VEL
LIN {X 0,Y 333.644,Z 431.925,A -85,B 0,C 180,E1 -14627.619,E2 -14627.619} C_VEL
LIN {X 0,Y 333.655,Z 431.924,A -85,B 0,C 180,E1 -14631.202,E2 -14631.202} C_VEL
LIN {X 0,Y 333.678,Z 431.917,A -85,B 0,C 180,E1 -14633.861,E2 -14633.861} C_VEL
LIN {X 0,Y 333.672,Z 431.962,A -85,B 0,C 180,E1 -14637.56,E2 -14637.56} C_VEL
LIN {X 0,Y 337.046,Z 445.118,A -85,B 0,C 180,E1 -14640.616,E2 -14640.616} C_VEL
LIN {X 0,Y 339.863,Z 458.936,A -85,B 0,C 180,E1 -14643.637,E2 -14643.637} C_VEL
LIN {X 0,Y 339.017,Z 472.991,A -85,B 0,C 180,E1 -14646.212,E2 -14646.212} C_VEL
LIN {X 0,Y 344.047,Z 501.046,A -85,B 0,C 180,E1 -14647.226,E2 -14647.226} C_VEL
LIN {X 0,Y 342.523,Z 579.802,A -85,B 0,C 180,E1 -14648.878,E2 -14648.878} C_VEL
LIN {X 0,Y 342.01,Z 593.171,A -85,B 0,C 180,E1 -14649.317,E2 -14649.317} C_VEL
LIN {X 0,Y 341.213,Z 605.894,A -85,B 0,C 180,E1 -14649.975,E2 -14649.975} C_VEL
LIN {X 0,Y 340.177,Z 618.119,A -85,B 0,C 180,E1 -14650.854,E2 -14650.854} C_VEL
LIN {X 0,Y 339.129,Z 629.024,A -85,B 0,C 180,E1 -14651.889,E2 -14651.889} C_VEL
LIN {X 0,Y 338.016,Z 639.03,A -85,B 0,C 180,E1 -14653.077,E2 -14653.077} C_VEL
LIN {X 0,Y 337.053,Z 647.29,A -85,B 0,C 180,E1 -14654.272,E2 -14654.272} C_VEL
LIN {X 0,Y 335.803,Z 655.878,A -85,B 0,C 180,E1 -14655.764,E2 -14655.764} C_VEL
LIN {X 0,Y 334.868,Z 662.963,A -85,B 0,C 180,E1 -14657.269,E2 -14657.269} C_VEL
LIN {X 0,Y 333.917,Z 669.923,A -85,B 0,C 180,E1 -14659.081,E2 -14659.081} C_VEL
LIN {X 0,Y 333.122,Z 675.453,A -85,B 0,C 180,E1 -14660.896,E2 -14660.896} C_VEL
LIN {X 0,Y 332.674,Z 679.789,A -85,B 0,C 180,E1 -14662.718,E2 -14662.718} C_VEL
LIN {X 0,Y 332.429,Z 682.07,A -85,B 0,C 180,E1 -14663.932,E2 -14663.932} C_VEL
LIN {X 0,Y 332.267,Z 683.93,A -85,B 0,C 180,E1 -14665.147,E2 -14665.147} C_VEL
LIN {X 0,Y 332.107,Z 685.351,A -85,B 0,C 180,E1 -14666.36,E2 -14666.36} C_VEL
LIN {X 0,Y 331.962,Z 686.961,A -85,B 0,C 180,E1 -14668.787,E2 -14668.787} C_VEL
LIN {X 0,Y 331.957,Z 687.194,A -85,B 0,C 180,E1 -14670,E2 -14670} C_VEL
LIN {X 0,Y 331.962,Z 687.001,A -85,B 0,C 180,E1 -14671.213,E2 -14671.213} C_VEL
LIN {X 0,Y 332.106,Z 685.445,A -85,B 0,C 180,E1 -14673.64,E2 -14673.64} C_VEL
LIN {X 0,Y 332.265,Z 684.077,A -85,B 0,C 180,E1 -14674.853,E2 -14674.853} C_VEL
LIN {X 0,Y 332.524,Z 681.331,A -85,B 0,C 180,E1 -14676.604,E2 -14676.604} C_VEL
LIN {X 0,Y 332.933,Z 677.297,A -85,B 0,C 180,E1 -14678.498,E2 -14678.498} C_VEL
LIN {X 0,Y 333.603,Z 672.232,A -85,B 0,C 180,E1 -14680.316,E2 -14680.316} C_VEL
LIN {X 0,Y 334.486,Z 665.846,A -85,B 0,C 180,E1 -14682.129,E2 -14682.129} C_VEL
LIN {X 0,Y 335.54,Z 657.912,A -85,B 0,C 180,E1 -14683.938,E2 -14683.938} C_VEL
LIN {X 0,Y 336.734,Z 649.796,A -85,B 0,C 180,E1 -14685.433,E2 -14685.433} C_VEL
LIN {X 0,Y 337.834,Z 640.982,A -85,B 0,C 180,E1 -14686.771,E2 -14686.771} C_VEL
LIN {X 0,Y 338.873,Z 631.34,A -85,B 0,C 180,E1 -14687.969,E2 -14687.969} C_VEL
LIN {X 0,Y 340.099,Z 619.277,A -85,B 0,C 180,E1 -14689.151,E2 -14689.151} C_VEL
LIN {X 0,Y 341.235,Z 607.531,A -85,B 0,C 180,E1 -14690.024,E2 -14690.024} C_VEL
LIN {X 0,Y 341.6,Z 601.893,A -85,B 0,C 180,E1 -14690.361,E2 -14690.361} C_VEL
LIN {X 0,Y 341.332,Z 596.308,A -85,B 0,C 180,E1 -14690.686,E2 -14690.686} C_VEL
LIN {X 0,Y 339.063,Z 587.196,A -85,B 0,C 180,E1 -14691.228,E2 -14691.228} C_VEL
LIN {X 0,Y 336.641,Z 577.947,A -85,B 0,C 180,E1 -14691.666,E2 -14691.666} C_VEL
LIN {X 0,Y 336.186,Z 572.153,A -85,B 0,C 180,E1 -14691.828,E2 -14691.828} C_VEL
LIN {X 0,Y 337.513,Z 502.096,A -85,B 0,C 180,E1 -14693.327,E2 -14693.327} C_VEL
LIN {X 0,Y 333.066,Z 476.974,A -85,B 0,C 180,E1 -14694.242,E2 -14694.242} C_VEL
LIN {X 0,Y 332.37,Z 473.145,A -85,B 0,C 180,E1 -14694.405,E2 -14694.405} C_VEL
LIN {X 0,Y 333.128,Z 461.458,A -85,B 0,C 180,E1 -14696.561,E2 -14696.561} C_VEL
LIN {X 0,Y 331.848,Z 454.301,A -85,B 0,C 180,E1 -14698.114,E2 -14698.114} C_VEL
LIN {X 0,Y 329.187,Z 442.46,A -85,B 0,C 180,E1 -14700.823,E2 -14700.823} C_VEL
LIN {X 0,Y 326.603,Z 432.805,A -85,B 0,C 180,E1 -14703.126,E2 -14703.126} C_VEL
LIN {X 0,Y 326.632,Z 432.797,A -85,B 0,C 180,E1 -14707.047,E2 -14707.047} C_VEL
LIN {X 0,Y 326.593,Z 432.796,A -85,B 0,C 180,E1 -14710.209,E2 -14710.209} C_VEL
LIN {X 0,Y 326.578,Z 432.797,A -85,B 0,C 180,E1 -14713.523,E2 -14713.523} C_VEL
LIN {X 0,Y 326.585,Z 432.801,A -85,B 0,C 180,E1 -14717.027,E2 -14717.027} C_VEL
LIN {X 0,Y 326.614,Z 432.805,A -85,B 0,C 180,E1 -14720.773,E2 -14720.773} C_VEL
LIN {X 0,Y 326.614,Z 432.787,A -85,B 0,C 180,E1 -14724.48,E2 -14724.48} C_VEL
LIN {X 0,Y 326.61,Z 432.801,A -85,B 0,C 180,E1 -14727.456,E2 -14727.456} C_VEL
LIN {X 0,Y 326.644,Z 432.834,A -85,B 0,C 180,E1 -14729.319,E2 -14729.319} C_VEL
LIN {X 0,Y 330.037,Z 448.766,A -85,B 0,C 180,E1 -14732.741,E2 -14732.741} C_VEL
LIN {X 0,Y 331.228,Z 455.807,A -85,B 0,C 180,E1 -14734.216,E2 -14734.216} C_VEL
LIN {X 0,Y 330.377,Z 469.131,A -85,B 0,C 180,E1 -14736.825,E2 -14736.825} C_VEL
LIN {X 0,Y 330.103,Z 473.904,A -85,B 0,C 180,E1 -14737.738,E2 -14737.738} C_VEL
LIN {X 0,Y 333.507,Z 501.731,A -85,B 0,C 180,E1 -14738.751,E2 -14738.751} C_VEL
LIN {X 0,Y 331.073,Z 585.1,A -85,B 0,C 180,E1 -14741.232,E2 -14741.232} C_VEL
LIN {X 0,Y 330.464,Z 598.694,A -85,B 0,C 180,E1 -14741.879,E2 -14741.879} C_VEL
LIN {X 0,Y 329.826,Z 610.352,A -85,B 0,C 180,E1 -14742.643,E2 -14742.643} C_VEL
LIN {X 0,Y 329.043,Z 622.812,A -85,B 0,C 180,E1 -14743.72,E2 -14743.72} C_VEL
LIN {X 0,Y 328.321,Z 633.748,A -85,B 0,C 180,E1 -14744.906,E2 -14744.906} C_VEL
LIN {X 0,Y 327.503,Z 644.418,A -85,B 0,C 180,E1 -14746.346,E2 -14746.346} C_VEL
LIN {X 0,Y 326.707,Z 653.809,A -85,B 0,C 180,E1 -14747.893,E2 -14747.893} C_VEL
LIN {X 0,Y 326.028,Z 662.893,A -85,B 0,C 180,E1 -14749.756,E2 -14749.756} C_VEL
LIN {X 0,Y 325.5,Z 670.222,A -85,B 0,C 180,E1 -14751.62,E2 -14751.62} C_VEL
LIN {X 0,Y 325.236,Z 675.156,A -85,B 0,C 180,E1 -14753.174,E2 -14753.174} C_VEL
LIN {X 0,Y 325.05,Z 679.873,A -85,B 0,C 180,E1 -14755.038,E2 -14755.038} C_VEL
LIN {X 0,Y 324.932,Z 683.396,A -85,B 0,C 180,E1 -14756.9,E2 -14756.9} C_VEL
LIN {X 0,Y 324.834,Z 685.845,A -85,B 0,C 180,E1 -14758.76,E2 -14758.76} C_VEL
LIN {X 0,Y 324.855,Z 686.911,A -85,B 0,C 180,E1 -14760,E2 -14760} C_VEL
LIN {X 0,Y 324.893,Z 687.55,A -85,B 0,C 180,E1 -14761.239,E2 -14761.239} C_VEL
LIN {X 0,Y 324.964,Z 687.706,A -85,B 0,C 180,E1 -14762.479,E2 -14762.479} C_VEL
LIN {X 0,Y 325.076,Z 687.446,A -85,B 0,C 180,E1 -14763.719,E2 -14763.719} C_VEL
LIN {X 0,Y 325.307,Z 686.766,A -85,B 0,C 180,E1 -14764.957,E2 -14764.957} C_VEL
LIN {X 0,Y 325.762,Z 684.551,A -85,B 0,C 180,E1 -14767.064,E2 -14767.064} C_VEL
LIN {X 0,Y 326.498,Z 680.778,A -85,B 0,C 180,E1 -14769.291,E2 -14769.291} C_VEL
LIN {X 0,Y 327.436,Z 676.426,A -85,B 0,C 180,E1 -14771.138,E2 -14771.138} C_VEL
LIN {X 0,Y 328.726,Z 669.782,A -85,B 0,C 180,E1 -14773.287,E2 -14773.287} C_VEL
LIN {X 0,Y 330.283,Z 662.521,A -85,B 0,C 180,E1 -14775.11,E2 -14775.11} C_VEL
LIN {X 0,Y 331.696,Z 655.119,A -85,B 0,C 180,E1 -14776.621,E2 -14776.621} C_VEL
LIN {X 0,Y 333.461,Z 645.877,A -85,B 0,C 180,E1 -14778.176,E2 -14778.176} C_VEL
LIN {X 0,Y 335.292,Z 635.509,A -85,B 0,C 180,E1 -14779.595,E2 -14779.595} C_VEL
LIN {X 0,Y 337.17,Z 623.34,A -85,B 0,C 180,E1 -14780.913,E2 -14780.913} C_VEL
LIN {X 0,Y 338.748,Z 611.474,A -85,B 0,C 180,E1 -14781.928,E2 -14781.928} C_VEL
LIN {X 0,Y 340.249,Z 598.419,A -85,B 0,C 180,E1 -14782.786,E2 -14782.786} C_VEL
LIN {X 0,Y 341.513,Z 584.713,A -85,B 0,C 180,E1 -14783.418,E2 -14783.418} C_VEL
LIN {X 0,Y 347.136,Z 511.304,A -85,B 0,C 180,E1 -14785.958,E2 -14785.958} C_VEL
LIN {X 0,Y 347.415,Z 506.402,A -85,B 0,C 180,E1 -14786.153,E2 -14786.153} C_VEL
LIN {X 0,Y 345.458,Z 494.582,A -85,B 0,C 180,E1 -14787.064,E2 -14787.064} C_VEL
LIN {X 0,Y 342.764,Z 481.978,A -85,B 0,C 180,E1 -14788.222,E2 -14788.222} C_VEL
LIN {X 0,Y 341.557,Z 476.98,A -85,B 0,C 180,E1 -14788.757,E2 -14788.757} C_VEL
LIN {X 0,Y 340.772,Z 470.188,A -85,B 0,C 180,E1 -14790.693,E2 -14790.693} C_VEL
LIN {X 0,Y 339.181,Z 462.777,A -85,B 0,C 180,E1 -14793.188,E2 -14793.188} C_VEL
LIN {X 0,Y 337.431,Z 456.56,A -85,B 0,C 180,E1 -14795.679,E2 -14795.679} C_VEL
LIN {X 0,Y 335.726,Z 451.635,A -85,B 0,C 180,E1 -14798.194,E2 -14798.194} C_VEL
LIN {X 0,Y 334.673,Z 449.024,A -85,B 0,C 180,E1 -14799.868,E2 -14799.868} C_VEL
LIN {X 0,Y 333.417,Z 446.087,A -85,B 0,C 180,E1 -14802.459,E2 -14802.459} C_VEL
LIN {X 0,Y 332.83,Z 444.944,A -85,B 0,C 180,E1 -14804.173,E2 -14804.173} C_VEL
LIN {X 0,Y 332.579,Z 444.238,A -85,B 0,C 180,E1 -14805.929,E2 -14805.929} C_VEL
LIN {X 0,Y 332.72,Z 444.175,A -85,B 0,C 180,E1 -14807.672,E2 -14807.672} C_VEL
LIN {X 0,Y 333.151,Z 444.821,A -85,B 0,C 180,E1 -14809.415,E2 -14809.415} C_VEL
LIN {X 0,Y 333.977,Z 446.035,A -85,B 0,C 180,E1 -14811.133,E2 -14811.133} C_VEL
LIN {X 0,Y 335.318,Z 447.624,A -85,B 0,C 180,E1 -14812.793,E2 -14812.793} C_VEL
LIN {X 0,Y 337.881,Z 452.112,A -85,B 0,C 180,E1 -14815.385,E2 -14815.385} C_VEL
LIN {X 0,Y 338.759,Z 453.772,A -85,B 0,C 180,E1 -14816.084,E2 -14816.084} C_VEL
LIN {X 0,Y 339.261,Z 457.021,A -85,B 0,C 180,E1 -14816.978,E2 -14816.978} C_VEL
LIN {X 0,Y 340.879,Z 467.023,A -85,B 0,C 180,E1 -14819.205,E2 -14819.205} C_VEL
LIN {X 0,Y 341.251,Z 469.591,A -85,B 0,C 180,E1 -14819.679,E2 -14819.679} C_VEL
LIN {X 0,Y 341.12,Z 481.489,A -85,B 0,C 180,E1 -14821.237,E2 -14821.237} C_VEL
LIN {X 0,Y 341.397,Z 484.768,A -85,B 0,C 180,E1 -14821.591,E2 -14821.591} C_VEL
LIN {X 0,Y 343.32,Z 499.828,A -85,B 0,C 180,E1 -14822.786,E2 -14822.786} C_VEL
LIN {X 0,Y 344.68,Z 514.904,A -85,B 0,C 180,E1 -14823.787,E2 -14823.787} C_VEL
LIN {X 0,Y 344.969,Z 531.844,A -85,B 0,C 180,E1 -14824.67,E2 -14824.67} C_VEL
LIN {X 0,Y 339.106,Z 607.511,A -85,B 0,C 180,E1 -14827.374,E2 -14827.374} C_VEL
LIN {X 0,Y 337.693,Z 620.69,A -85,B 0,C 180,E1 -14828.08,E2 -14828.08} C_VEL
LIN {X 0,Y 336.037,Z 633.419,A -85,B 0,C 180,E1 -14829.013,E2 -14829.013} C_VEL
LIN {X 0,Y 334.183,Z 645.7,A -85,B 0,C 180,E1 -14830.177,E2 -14830.177} C_VEL
LIN {X 0,Y 332.439,Z 656.765,A -85,B 0,C 180,E1 -14831.512,E2 -14831.512} C_VEL
LIN {X 0,Y 330.782,Z 666.784,A -85,B 0,C 180,E1 -14833.031,E2 -14833.031} C_VEL
LIN {X 0,Y 328.988,Z 676.471,A -85,B 0,C 180,E1 -14834.83,E2 -14834.83} C_VEL
LIN {X 0,Y 327.646,Z 684.276,A -85,B 0,C 180,E1 -14836.668,E2 -14836.668} C_VEL
LIN {X 0,Y 326.734,Z 689.612,A -85,B 0,C 180,E1 -14838.209,E2 -14838.209} C_VEL
LIN {X 0,Y 325.946,Z 694.781,A -85,B 0,C 180,E1 -14840.067,E2 -14840.067} C_VEL
LIN {X 0,Y 325.374,Z 698.776,A -85,B 0,C 180,E1 -14841.929,E2 -14841.929} C_VEL
LIN {X 0,Y 325.037,Z 701.995,A -85,B 0,C 180,E1 -14844.055,E2 -14844.055} C_VEL
LIN {X 0,Y 324.957,Z 703.886,A -85,B 0,C 180,E1 -14846.28,E2 -14846.28} C_VEL
LIN {X 0,Y 324.944,Z 704.692,A -85,B 0,C 180,E1 -14850,E2 -14850} C_VEL
LIN {X 0,Y 324.886,Z 704.466,A -85,B 0,C 180,E1 -14851.24,E2 -14851.24} C_VEL
LIN {X 0,Y 324.894,Z 703.847,A -85,B 0,C 180,E1 -14852.48,E2 -14852.48} C_VEL
LIN {X 0,Y 324.953,Z 702.837,A -85,B 0,C 180,E1 -14853.72,E2 -14853.72} C_VEL
LIN {X 0,Y 325.001,Z 700.054,A -85,B 0,C 180,E1 -14855.884,E2 -14855.884} C_VEL
LIN {X 0,Y 325.292,Z 695.819,A -85,B 0,C 180,E1 -14858.073,E2 -14858.073} C_VEL
LIN {X 0,Y 325.772,Z 691.002,A -85,B 0,C 180,E1 -14859.938,E2 -14859.938} C_VEL
LIN {X 0,Y 326.416,Z 684.905,A -85,B 0,C 180,E1 -14861.803,E2 -14861.803} C_VEL
LIN {X 0,Y 327.486,Z 677.309,A -85,B 0,C 180,E1 -14863.654,E2 -14863.654} C_VEL
LIN {X 0,Y 328.668,Z 668.307,A -85,B 0,C 180,E1 -14865.398,E2 -14865.398} C_VEL
LIN {X 0,Y 329.922,Z 657.817,A -85,B 0,C 180,E1 -14867.032,E2 -14867.032} C_VEL
LIN {X 0,Y 331.33,Z 646.607,A -85,B 0,C 180,E1 -14868.392,E2 -14868.392} C_VEL
LIN {X 0,Y 332.207,Z 639.505,A -85,B 0,C 180,E1 -14869.142,E2 -14869.142} C_VEL
LIN {X 0,Y 334.48,Z 626.675,A -85,B 0,C 180,E1 -14870.606,E2 -14870.606} C_VEL
LIN {X 0,Y 336.68,Z 613.868,A -85,B 0,C 180,E1 -14871.748,E2 -14871.748} C_VEL
LIN {X 0,Y 338.784,Z 599.357,A -85,B 0,C 180,E1 -14872.729,E2 -14872.729} C_VEL
LIN {X 0,Y 340.375,Z 585.277,A -85,B 0,C 180,E1 -14873.42,E2 -14873.42} C_VEL
LIN {X 0,Y 344.385,Z 528.538,A -85,B 0,C 180,E1 -14875.398,E2 -14875.398} C_VEL
LIN {X 0,Y 343.791,Z 514.852,A -85,B 0,C 180,E1 -14876.119,E2 -14876.119} C_VEL
LIN {X 0,Y 342.354,Z 500.733,A -85,B 0,C 180,E1 -14877.029,E2 -14877.029} C_VEL
LIN {X 0,Y 340.209,Z 487.066,A -85,B 0,C 180,E1 -14878.097,E2 -14878.097} C_VEL
LIN {X 0,Y 337.281,Z 472.363,A -85,B 0,C 180,E1 -14879.462,E2 -14879.462} C_VEL
LIN {X 0,Y 336,Z 467.498,A -85,B 0,C 180,E1 -14880.058,E2 -14880.058} C_VEL
LIN {X 0,Y 335.04,Z 461.597,A -85,B 0,C 180,E1 -14882.035,E2 -14882.035} C_VEL
LIN {X 0,Y 333.515,Z 454.591,A -85,B 0,C 180,E1 -14884.731,E2 -14884.731} C_VEL
LIN {X 0,Y 332.118,Z 449.474,A -85,B 0,C 180,E1 -14887.091,E2 -14887.091} C_VEL
LIN {X 0,Y 330.726,Z 444.985,A -85,B 0,C 180,E1 -14889.606,E2 -14889.606} C_VEL
LIN {X 0,Y 329.712,Z 441.873,A -85,B 0,C 180,E1 -14891.751,E2 -14891.751} C_VEL
LIN {X 0,Y 328.473,Z 438.404,A -85,B 0,C 180,E1 -14895.084,E2 -14895.084} C_VEL
LIN {X 0,Y 327.743,Z 436.381,A -85,B 0,C 180,E1 -14898.636,E2 -14898.636} C_VEL
LIN {X 0,Y 327.681,Z 435.9,A -85,B 0,C 180,E1 -14901.539,E2 -14901.539} C_VEL
LIN {X 0,Y 327.824,Z 436.66,A -85,B 0,C 180,E1 -14904.631,E2 -14904.631} C_VEL
LIN {X 0,Y 328.45,Z 438.421,A -85,B 0,C 180,E1 -14907.66,E2 -14907.66} C_VEL
LIN {X 0,Y 328.676,Z 439.096,A -85,B 0,C 180,E1 -14908.304,E2 -14908.304} C_VEL
LIN {X 0,Y 330.938,Z 442.047,A -85,B 0,C 180,E1 -14909.179,E2 -14909.179} C_VEL
LIN {X 0,Y 332.616,Z 443.786,A -85,B 0,C 180,E1 -14909.739,E2 -14909.739} C_VEL
LIN {X 0,Y 336.302,Z 448.599,A -85,B 0,C 180,E1 -14910.96,E2 -14910.96} C_VEL
LIN {X 0,Y 338.855,Z 451.985,A -85,B 0,C 180,E1 -14911.713,E2 -14911.713} C_VEL
LIN {X 0,Y 342.929,Z 458.059,A -85,B 0,C 180,E1 -14912.878,E2 -14912.878} C_VEL
LIN {X 0,Y 346.756,Z 465.286,A -85,B 0,C 180,E1 -14913.952,E2 -14913.952} C_VEL
LIN {X 0,Y 347.962,Z 467.874,A -85,B 0,C 180,E1 -14914.277,E2 -14914.277} C_VEL
LIN {X 0,Y 342.906,Z 531.301,A -85,B 0,C 180,E1 -14916.523,E2 -14916.523} C_VEL
LIN {X 0,Y 341.97,Z 545.444,A -85,B 0,C 180,E1 -14917.175,E2 -14917.175} C_VEL
LIN {X 0,Y 341.009,Z 556.729,A -85,B 0,C 180,E1 -14917.906,E2 -14917.906} C_VEL
LIN {X 0,Y 339.53,Z 569.287,A -85,B 0,C 180,E1 -14918.961,E2 -14918.961} C_VEL
LIN {X 0,Y 337.766,Z 581.411,A -85,B 0,C 180,E1 -14920.257,E2 -14920.257} C_VEL
LIN {X 0,Y 335.929,Z 592.189,A -85,B 0,C 180,E1 -14921.711,E2 -14921.711} C_VEL
LIN {X 0,Y 334.347,Z 601.03,A -85,B 0,C 180,E1 -14923.2,E2 -14923.2} C_VEL
LIN {X 0,Y 332.559,Z 609.598,A -85,B 0,C 180,E1 -14924.996,E2 -14924.996} C_VEL
LIN {X 0,Y 330.991,Z 616.574,A -85,B 0,C 180,E1 -14926.806,E2 -14926.806} C_VEL
LIN {X 0,Y 329.571,Z 622.52,A -85,B 0,C 180,E1 -14928.795,E2 -14928.795} C_VEL
LIN {X 0,Y 328.338,Z 626.939,A -85,B 0,C 180,E1 -14930.762,E2 -14930.762} C_VEL
LIN {X 0,Y 327.413,Z 629.924,A -85,B 0,C 180,E1 -14932.6,E2 -14932.6} C_VEL
LIN {X 0,Y 326.986,Z 631.344,A -85,B 0,C 180,E1 -14933.831,E2 -14933.831} C_VEL
LIN {X 0,Y 326.557,Z 632.346,A -85,B 0,C 180,E1 -14935.062,E2 -14935.062} C_VEL
LIN {X 0,Y 326.143,Z 632.881,A -85,B 0,C 180,E1 -14936.293,E2 -14936.293} C_VEL
LIN {X 0,Y 325.835,Z 632.994,A -85,B 0,C 180,E1 -14937.528,E2 -14937.528} C_VEL
LIN {X 0,Y 325.663,Z 632.683,A -85,B 0,C 180,E1 -14938.763,E2 -14938.763} C_VEL
LIN {X 0,Y 325.584,Z 631.919,A -85,B 0,C 180,E1 -14940,E2 -14940} C_VEL
LIN {X 0,Y 325.564,Z 630.716,A -85,B 0,C 180,E1 -14941.237,E2 -14941.237} C_VEL
LIN {X 0,Y 325.689,Z 628.096,A -85,B 0,C 180,E1 -14943.093,E2 -14943.093} C_VEL
LIN {X 0,Y 325.884,Z 624.421,A -85,B 0,C 180,E1 -14944.949,E2 -14944.949} C_VEL
LIN {X 0,Y 326.067,Z 619.594,A -85,B 0,C 180,E1 -14946.808,E2 -14946.808} C_VEL
LIN {X 0,Y 326.379,Z 613.478,A -85,B 0,C 180,E1 -14948.669,E2 -14948.669} C_VEL
LIN {X 0,Y 326.922,Z 605.828,A -85,B 0,C 180,E1 -14950.529,E2 -14950.529} C_VEL
LIN {X 0,Y 327.635,Z 596.317,A -85,B 0,C 180,E1 -14952.387,E2 -14952.387} C_VEL
LIN {X 0,Y 328.376,Z 586.549,A -85,B 0,C 180,E1 -14953.932,E2 -14953.932} C_VEL
LIN {X 0,Y 329.204,Z 574.415,A -85,B 0,C 180,E1 -14955.477,E2 -14955.477} C_VEL
LIN {X 0,Y 329.928,Z 563.135,A -85,B 0,C 180,E1 -14956.621,E2 -14956.621} C_VEL
LIN {X 0,Y 330.539,Z 549.284,A -85,B 0,C 180,E1 -14957.717,E2 -14957.717} C_VEL
LIN {X 0,Y 331.145,Z 535.96,A -85,B 0,C 180,E1 -14958.483,E2 -14958.483} C_VEL
LIN {X 0,Y 331.482,Z 522.247,A -85,B 0,C 180,E1 -14959.025,E2 -14959.025} C_VEL
LIN {X 0,Y 333.368,Z 453.714,A -85,B 0,C 180,E1 -14961.056,E2 -14961.056} C_VEL
LIN {X 0,Y 326.625,Z 432.796,A -85,B 0,C 180,E1 -14962.028,E2 -14962.028} C_VEL
LIN {X 0,Y 326.692,Z 432.793,A -85,B 0,C 180,E1 -14965.484,E2 -14965.484} C_VEL
LIN {X 0,Y 326.65,Z 432.797,A -85,B 0,C 180,E1 -14969.66,E2 -14969.66} C_VEL
LIN {X 0,Y 326.609,Z 432.775,A -85,B 0,C 180,E1 -14974.019,E2 -14974.019} C_VEL
LIN {X 0,Y 326.63,Z 432.803,A -85,B 0,C 180,E1 -14977.239,E2 -14977.239} C_VEL
LIN {X 0,Y 326.579,Z 432.791,A -85,B 0,C 180,E1 -14981.131,E2 -14981.131} C_VEL
LIN {X 0,Y 326.53,Z 432.804,A -85,B 0,C 180,E1 -14984.743,E2 -14984.743} C_VEL
LIN {X 0,Y 326.578,Z 432.806,A -85,B 0,C 180,E1 -14988.154,E2 -14988.154} C_VEL
LIN {X 0,Y 326.625,Z 432.801,A -85,B 0,C 180,E1 -14991.391,E2 -14991.391} C_VEL
LIN {X 0,Y 326.622,Z 432.801,A -85,B 0,C 180,E1 -14994.851,E2 -14994.851} C_VEL
LIN {X 0,Y 326.637,Z 432.973,A -85,B 0,C 180,E1 -14997.049,E2 -14997.049} C_VEL
LIN {X 0,Y 329.853,Z 445.162,A -85,B 0,C 180,E1 -14999.954,E2 -14999.954} C_VEL
LIN {X 0,Y 332.926,Z 459.624,A -85,B 0,C 180,E1 -15003.179,E2 -15003.179} C_VEL
LIN {X 0,Y 332.949,Z 463.939,A -85,B 0,C 180,E1 -15004.024,E2 -15004.024} C_VEL
LIN {X 0,Y 332.347,Z 473.196,A -85,B 0,C 180,E1 -15005.715,E2 -15005.715} C_VEL
LIN {X 0,Y 337.529,Z 502.133,A -85,B 0,C 180,E1 -15006.784,E2 -15006.784} C_VEL
LIN {X 0,Y 335.934,Z 579.913,A -85,B 0,C 180,E1 -15008.443,E2 -15008.443} C_VEL
LIN {X 0,Y 335.401,Z 593.324,A -85,B 0,C 180,E1 -15008.891,E2 -15008.891} C_VEL
LIN {X 0,Y 334.572,Z 606.061,A -85,B 0,C 180,E1 -15009.56,E2 -15009.56} C_VEL
LIN {X 0,Y 333.477,Z 618.295,A -85,B 0,C 180,E1 -15010.454,E2 -15010.454} C_VEL
LIN {X 0,Y 332.197,Z 630.58,A -85,B 0,C 180,E1 -15011.657,E2 -15011.657} C_VEL
LIN {X 0,Y 331.011,Z 641.487,A -85,B 0,C 180,E1 -15013.031,E2 -15013.031} C_VEL
LIN {X 0,Y 329.693,Z 651.113,A -85,B 0,C 180,E1 -15014.546,E2 -15014.546} C_VEL
LIN {X 0,Y 328.231,Z 660.498,A -85,B 0,C 180,E1 -15016.377,E2 -15016.377} C_VEL
LIN {X 0,Y 327.24,Z 667.944,A -85,B 0,C 180,E1 -15018.227,E2 -15018.227} C_VEL
LIN {X 0,Y 326.363,Z 673.921,A -85,B 0,C 180,E1 -15020.08,E2 -15020.08} C_VEL
LIN {X 0,Y 325.758,Z 678.646,A -85,B 0,C 180,E1 -15021.939,E2 -15021.939} C_VEL
LIN {X 0,Y 325.37,Z 682.259,A -85,B 0,C 180,E1 -15023.8,E2 -15023.8} C_VEL
LIN {X 0,Y 325.194,Z 684.119,A -85,B 0,C 180,E1 -15025.041,E2 -15025.041} C_VEL
LIN {X 0,Y 325.04,Z 685.54,A -85,B 0,C 180,E1 -15026.281,E2 -15026.281} C_VEL
LIN {X 0,Y 324.87,Z 687.15,A -85,B 0,C 180,E1 -15028.76,E2 -15028.76} C_VEL
LIN {X 0,Y 324.863,Z 687.383,A -85,B 0,C 180,E1 -15030,E2 -15030} C_VEL
LIN {X 0,Y 324.87,Z 687.19,A -85,B 0,C 180,E1 -15031.24,E2 -15031.24} C_VEL
LIN {X 0,Y 325.039,Z 685.633,A -85,B 0,C 180,E1 -15033.719,E2 -15033.719} C_VEL
LIN {X 0,Y 325.192,Z 684.265,A -85,B 0,C 180,E1 -15034.959,E2 -15034.959} C_VEL
LIN {X 0,Y 325.449,Z 681.76,A -85,B 0,C 180,E1 -15036.604,E2 -15036.604} C_VEL
LIN {X 0,Y 325.898,Z 677.484,A -85,B 0,C 180,E1 -15038.682,E2 -15038.682} C_VEL
LIN {X 0,Y 326.622,Z 672.418,A -85,B 0,C 180,E1 -15040.539,E2 -15040.539} C_VEL
LIN {X 0,Y 327.547,Z 666.03,A -85,B 0,C 180,E1 -15042.39,E2 -15042.39} C_VEL
LIN {X 0,Y 328.655,Z 658.094,A -85,B 0,C 180,E1 -15044.236,E2 -15044.236} C_VEL
LIN {X 0,Y 329.893,Z 649.976,A -85,B 0,C 180,E1 -15045.761,E2 -15045.761} C_VEL
LIN {X 0,Y 331.062,Z 640.651,A -85,B 0,C 180,E1 -15047.197,E2 -15047.197} C_VEL
LIN {X 0,Y 332.294,Z 630.136,A -85,B 0,C 180,E1 -15048.497,E2 -15048.497} C_VEL
LIN {X 0,Y 333.411,Z 619.442,A -85,B 0,C 180,E1 -15049.55,E2 -15049.55} C_VEL
LIN {X 0,Y 334.573,Z 607.685,A -85,B 0,C 180,E1 -15050.44,E2 -15050.44} C_VEL
LIN {X 0,Y 335.34,Z 594.753,A -85,B 0,C 180,E1 -15051.154,E2 -15051.154} C_VEL
LIN {X 0,Y 335.896,Z 582.303,A -85,B 0,C 180,E1 -15051.6,E2 -15051.6} C_VEL
LIN {X 0,Y 336.186,Z 572.153,A -85,B 0,C 180,E1 -15051.828,E2 -15051.828} C_VEL
LIN {X 0,Y 335.782,Z 566.342,A -85,B 0,C 180,E1 -15051.988,E2 -15051.988} C_VEL
LIN {X 0,Y 330.858,Z 547.653,A -85,B 0,C 180,E1 -15052.766,E2 -15052.766} C_VEL
LIN {X 0,Y 330.329,Z 541.842,A -85,B 0,C 180,E1 -15052.94,E2 -15052.94} C_VEL
LIN {X 0,Y 330.968,Z 502.757,A -85,B 0,C 180,E1 -15053.802,E2 -15053.802} C_VEL
LIN {X 0,Y 326.315,Z 476.598,A -85,B 0,C 180,E1 -15054.787,E2 -15054.787} C_VEL
LIN {X 0,Y 325.702,Z 473.237,A -85,B 0,C 180,E1 -15054.94,E2 -15054.94} C_VEL
LIN {X 0,Y 326.345,Z 462.811,A -85,B 0,C 180,E1 -15056.888,E2 -15056.888} C_VEL
LIN {X 0,Y 324.151,Z 451.482,A -85,B 0,C 180,E1 -15059.408,E2 -15059.408} C_VEL
LIN {X 0,Y 321.355,Z 440.34,A -85,B 0,C 180,E1 -15062.029,E2 -15062.029} C_VEL
LIN {X 0,Y 319.57,Z 433.685,A -85,B 0,C 180,E1 -15063.731,E2 -15063.731} C_VEL
LIN {X 0,Y 319.561,Z 433.683,A -85,B 0,C 180,E1 -15066.428,E2 -15066.428} C_VEL
LIN {X 0,Y 319.56,Z 433.674,A -85,B 0,C 180,E1 -15069.669,E2 -15069.669} C_VEL
LIN {X 0,Y 319.559,Z 433.672,A -85,B 0,C 180,E1 -15073.467,E2 -15073.467} C_VEL
LIN {X 0,Y 319.564,Z 433.675,A -85,B 0,C 180,E1 -15077.018,E2 -15077.018} C_VEL
LIN {X 0,Y 319.549,Z 433.682,A -85,B 0,C 180,E1 -15080.371,E2 -15080.371} C_VEL
LIN {X 0,Y 319.561,Z 433.661,A -85,B 0,C 180,E1 -15083.572,E2 -15083.572} C_VEL
LIN {X 0,Y 319.579,Z 433.679,A -85,B 0,C 180,E1 -15086.686,E2 -15086.686} C_VEL
LIN {X 0,Y 319.609,Z 433.693,A -85,B 0,C 180,E1 -15089.047,E2 -15089.047} C_VEL
LIN {X 0,Y 322.896,Z 449.302,A -85,B 0,C 180,E1 -15092.45,E2 -15092.45} C_VEL
LIN {X 0,Y 324.22,Z 456.414,A -85,B 0,C 180,E1 -15093.963,E2 -15093.963} C_VEL
LIN {X 0,Y 323.525,Z 468.273,A -85,B 0,C 180,E1 -15096.316,E2 -15096.316} C_VEL
LIN {X 0,Y 323.201,Z 474.151,A -85,B 0,C 180,E1 -15097.444,E2 -15097.444} C_VEL
LIN {X 0,Y 326.375,Z 499.597,A -85,B 0,C 180,E1 -15098.393,E2 -15098.393} C_VEL
LIN {X 0,Y 326.549,Z 503.931,A -85,B 0,C 180,E1 -15098.538,E2 -15098.538} C_VEL
LIN {X 0,Y 324.037,Z 585.273,A -85,B 0,C 180,E1 -15101.055,E2 -15101.055} C_VEL
LIN {X 0,Y 323.431,Z 598.765,A -85,B 0,C 180,E1 -15101.716,E2 -15101.716} C_VEL
LIN {X 0,Y 322.688,Z 611.372,A -85,B 0,C 180,E1 -15102.574,E2 -15102.574} C_VEL
LIN {X 0,Y 321.867,Z 624.069,A -85,B 0,C 180,E1 -15103.713,E2 -15103.713} C_VEL
LIN {X 0,Y 321.197,Z 634.879,A -85,B 0,C 180,E1 -15104.94,E2 -15104.94} C_VEL
LIN {X 0,Y 320.3,Z 646.112,A -85,B 0,C 180,E1 -15106.518,E2 -15106.518} C_VEL
LIN {X 0,Y 319.434,Z 656.011,A -85,B 0,C 180,E1 -15108.257,E2 -15108.257} C_VEL
LIN {X 0,Y 318.789,Z 664.764,A -85,B 0,C 180,E1 -15110.162,E2 -15110.162} C_VEL
LIN {X 0,Y 318.338,Z 671.728,A -85,B 0,C 180,E1 -15112.069,E2 -15112.069} C_VEL
LIN {X 0,Y 318.036,Z 677.197,A -85,B 0,C 180,E1 -15113.944,E2 -15113.944} C_VEL
LIN {X 0,Y 317.956,Z 680.914,A -85,B 0,C 180,E1 -15115.563,E2 -15115.563} C_VEL
LIN {X 0,Y 317.809,Z 684.213,A -85,B 0,C 180,E1 -15117.465,E2 -15117.465} C_VEL
LIN {X 0,Y 317.747,Z 685.833,A -85,B 0,C 180,E1 -15118.733,E2 -15118.733} C_VEL
LIN {X 0,Y 317.764,Z 686.959,A -85,B 0,C 180,E1 -15120,E2 -15120} C_VEL
LIN {X 0,Y 317.804,Z 687.672,A -85,B 0,C 180,E1 -15121.267,E2 -15121.267} C_VEL
LIN {X 0,Y 317.883,Z 687.951,A -85,B 0,C 180,E1 -15122.534,E2 -15122.534} C_VEL
LIN {X 0,Y 318.013,Z 687.755,A -85,B 0,C 180,E1 -15123.801,E2 -15123.801} C_VEL
LIN {X 0,Y 318.265,Z 687.145,A -85,B 0,C 180,E1 -15125.067,E2 -15125.067} C_VEL
LIN {X 0,Y 318.729,Z 685.211,A -85,B 0,C 180,E1 -15127.134,E2 -15127.134} C_VEL
LIN {X 0,Y 319.54,Z 681.505,A -85,B 0,C 180,E1 -15129.495,E2 -15129.495} C_VEL
LIN {X 0,Y 320.531,Z 677.306,A -85,B 0,C 180,E1 -15131.381,E2 -15131.381} C_VEL
LIN {X 0,Y 321.65,Z 671.91,A -85,B 0,C 180,E1 -15133.263,E2 -15133.263} C_VEL
LIN {X 0,Y 323.247,Z 665.12,A -85,B 0,C 180,E1 -15135.124,E2 -15135.124} C_VEL
LIN {X 0,Y 325.062,Z 656.723,A -85,B 0,C 180,E1 -15136.97,E2 -15136.97} C_VEL
LIN {X 0,Y 327.036,Z 647.257,A -85,B 0,C 180,E1 -15138.633,E2 -15138.633} C_VEL
LIN {X 0,Y 329.25,Z 635.413,A -85,B 0,C 180,E1 -15140.296,E2 -15140.296} C_VEL
LIN {X 0,Y 331.296,Z 623.332,A -85,B 0,C 180,E1 -15141.629,E2 -15141.629} C_VEL
LIN {X 0,Y 333,Z 611.495,A -85,B 0,C 180,E1 -15142.654,E2 -15142.654} C_VEL
LIN {X 0,Y 334.574,Z 598.396,A -85,B 0,C 180,E1 -15143.523,E2 -15143.523} C_VEL
LIN {X 0,Y 336.076,Z 582.891,A -85,B 0,C 180,E1 -15144.23,E2 -15144.23} C_VEL
LIN {X 0,Y 342.29,Z 508.601,A -85,B 0,C 180,E1 -15146.887,E2 -15146.887} C_VEL
LIN {X 0,Y 340.518,Z 497.148,A -85,B 0,C 180,E1 -15147.81,E2 -15147.81} C_VEL
LIN {X 0,Y 338.05,Z 484.788,A -85,B 0,C 180,E1 -15149.002,E2 -15149.002} C_VEL
LIN {X 0,Y 336.971,Z 480.702,A -85,B 0,C 180,E1 -15149.481,E2 -15149.481} C_VEL
LIN {X 0,Y 335.554,Z 477.183,A -85,B 0,C 180,E1 -15150.07,E2 -15150.07} C_VEL
LIN {X 0,Y 334.595,Z 471.125,A -85,B 0,C 180,E1 -15152.014,E2 -15152.014} C_VEL
LIN {X 0,Y 333.086,Z 464.192,A -85,B 0,C 180,E1 -15154.625,E2 -15154.625} C_VEL
LIN {X 0,Y 331.477,Z 458.542,A -85,B 0,C 180,E1 -15157.274,E2 -15157.274} C_VEL
LIN {X 0,Y 329.978,Z 454.336,A -85,B 0,C 180,E1 -15159.937,E2 -15159.937} C_VEL
LIN {X 0,Y 329.199,Z 452.421,A -85,B 0,C 180,E1 -15161.651,E2 -15161.651} C_VEL
LIN {X 0,Y 328.667,Z 451.059,A -85,B 0,C 180,E1 -15163.361,E2 -15163.361} C_VEL
LIN {X 0,Y 328.375,Z 450.221,A -85,B 0,C 180,E1 -15165.067,E2 -15165.067} C_VEL
LIN {X 0,Y 328.412,Z 449.896,A -85,B 0,C 180,E1 -15166.78,E2 -15166.78} C_VEL
LIN {X 0,Y 328.732,Z 450.2,A -85,B 0,C 180,E1 -15168.49,E2 -15168.49} C_VEL
LIN {X 0,Y 329.437,Z 451.176,A -85,B 0,C 180,E1 -15170.208,E2 -15170.208} C_VEL
LIN {X 0,Y 331.365,Z 453.626,A -85,B 0,C 180,E1 -15172.809,E2 -15172.809} C_VEL
LIN {X 0,Y 333.96,Z 458.156,A -85,B 0,C 180,E1 -15175.375,E2 -15175.375} C_VEL
LIN {X 0,Y 334.622,Z 460.085,A -85,B 0,C 180,E1 -15176.074,E2 -15176.074} C_VEL
LIN {X 0,Y 336,Z 470.312,A -85,B 0,C 180,E1 -15178.472,E2 -15178.472} C_VEL
LIN {X 0,Y 336.4,Z 473.541,A -85,B 0,C 180,E1 -15179.094,E2 -15179.094} C_VEL
LIN {X 0,Y 336.16,Z 483.518,A -85,B 0,C 180,E1 -15180.424,E2 -15180.424} C_VEL
LIN {X 0,Y 337.951,Z 497.287,A -85,B 0,C 180,E1 -15181.641,E2 -15181.641} C_VEL
LIN {X 0,Y 339.325,Z 512.708,A -85,B 0,C 180,E1 -15182.767,E2 -15182.767} C_VEL
LIN {X 0,Y 339.69,Z 523.87,A -85,B 0,C 180,E1 -15183.418,E2 -15183.418} C_VEL
LIN {X 0,Y 339.667,Z 533.167,A -85,B 0,C 180,E1 -15183.902,E2 -15183.902} C_VEL
LIN {X 0,Y 333.422,Z 607.21,A -85,B 0,C 180,E1 -15186.638,E2 -15186.638} C_VEL
LIN {X 0,Y 331.76,Z 621.32,A -85,B 0,C 180,E1 -15187.421,E2 -15187.421} C_VEL
LIN {X 0,Y 330.147,Z 632.994,A -85,B 0,C 180,E1 -15188.292,E2 -15188.292} C_VEL
LIN {X 0,Y 328.18,Z 645.199,A -85,B 0,C 180,E1 -15189.471,E2 -15189.471} C_VEL
LIN {X 0,Y 326.26,Z 656.191,A -85,B 0,C 180,E1 -15190.822,E2 -15190.822} C_VEL
LIN {X 0,Y 324.361,Z 666.692,A -85,B 0,C 180,E1 -15192.432,E2 -15192.432} C_VEL
LIN {X 0,Y 322.5,Z 675.992,A -85,B 0,C 180,E1 -15194.193,E2 -15194.193} C_VEL
LIN {X 0,Y 320.955,Z 683.796,A -85,B 0,C 180,E1 -15196.062,E2 -15196.062} C_VEL
LIN {X 0,Y 319.811,Z 690.134,A -85,B 0,C 180,E1 -15197.95,E2 -15197.95} C_VEL
LIN {X 0,Y 318.961,Z 695.151,A -85,B 0,C 180,E1 -15199.847,E2 -15199.847} C_VEL
LIN {X 0,Y 318.338,Z 698.978,A -85,B 0,C 180,E1 -15201.749,E2 -15201.749} C_VEL
LIN {X 0,Y 317.95,Z 702.192,A -85,B 0,C 180,E1 -15204.091,E2 -15204.091} C_VEL
LIN {X 0,Y 317.863,Z 703.769,A -85,B 0,C 180,E1 -15206.197,E2 -15206.197} C_VEL
LIN {X 0,Y 317.849,Z 704.503,A -85,B 0,C 180,E1 -15210,E2 -15210} C_VEL
LIN {X 0,Y 317.795,Z 704.277,A -85,B 0,C 180,E1 -15211.267,E2 -15211.267} C_VEL
LIN {X 0,Y 317.813,Z 703.658,A -85,B 0,C 180,E1 -15212.535,E2 -15212.535} C_VEL
LIN {X 0,Y 317.859,Z 702.648,A -85,B 0,C 180,E1 -15213.803,E2 -15213.803} C_VEL
LIN {X 0,Y 317.894,Z 700.173,A -85,B 0,C 180,E1 -15215.81,E2 -15215.81} C_VEL
LIN {X 0,Y 318.116,Z 696.984,A -85,B 0,C 180,E1 -15217.617,E2 -15217.617} C_VEL
LIN {X 0,Y 318.549,Z 692.563,A -85,B 0,C 180,E1 -15219.525,E2 -15219.525} C_VEL
LIN {X 0,Y 319.166,Z 686.927,A -85,B 0,C 180,E1 -15221.431,E2 -15221.431} C_VEL
LIN {X 0,Y 320.183,Z 679.834,A -85,B 0,C 180,E1 -15223.325,E2 -15223.325} C_VEL
LIN {X 0,Y 321.367,Z 670.973,A -85,B 0,C 180,E1 -15225.214,E2 -15225.214} C_VEL
LIN {X 0,Y 322.605,Z 661.866,A -85,B 0,C 180,E1 -15226.777,E2 -15226.777} C_VEL
LIN {X 0,Y 323.905,Z 651.727,A -85,B 0,C 180,E1 -15228.174,E2 -15228.174} C_VEL
LIN {X 0,Y 325.157,Z 642.689,A -85,B 0,C 180,E1 -15229.246,E2 -15229.246} C_VEL
LIN {X 0,Y 327.484,Z 630.901,A -85,B 0,C 180,E1 -15230.738,E2 -15230.738} C_VEL
LIN {X 0,Y 329.595,Z 619.446,A -85,B 0,C 180,E1 -15231.91,E2 -15231.91} C_VEL
LIN {X 0,Y 331.918,Z 605.886,A -85,B 0,C 180,E1 -15232.979,E2 -15232.979} C_VEL
LIN {X 0,Y 333.792,Z 593.15,A -85,B 0,C 180,E1 -15233.746,E2 -15233.746} C_VEL
LIN {X 0,Y 335.128,Z 579.984,A -85,B 0,C 180,E1 -15234.344,E2 -15234.344} C_VEL
LIN {X 0,Y 338.929,Z 529.526,A -85,B 0,C 180,E1 -15236.146,E2 -15236.146} C_VEL
LIN {X 0,Y 338.469,Z 516.272,A -85,B 0,C 180,E1 -15236.874,E2 -15236.874} C_VEL
LIN {X 0,Y 337.172,Z 502.417,A -85,B 0,C 180,E1 -15237.811,E2 -15237.811} C_VEL
LIN {X 0,Y 335.241,Z 489.17,A -85,B 0,C 180,E1 -15238.896,E2 -15238.896} C_VEL
LIN {X 0,Y 332.646,Z 475.398,A -85,B 0,C 180,E1 -15240.245,E2 -15240.245} C_VEL
LIN {X 0,Y 331.579,Z 471.745,A -85,B 0,C 180,E1 -15240.714,E2 -15240.714} C_VEL
LIN {X 0,Y 328.825,Z 465.479,A -85,B 0,C 180,E1 -15241.84,E2 -15241.84} C_VEL
LIN {X 0,Y 327.482,Z 458.974,A -85,B 0,C 180,E1 -15244.363,E2 -15244.363} C_VEL
LIN {X 0,Y 325.973,Z 453.023,A -85,B 0,C 180,E1 -15247.134,E2 -15247.134} C_VEL
LIN {X 0,Y 324.577,Z 448.447,A -85,B 0,C 180,E1 -15249.766,E2 -15249.766} C_VEL
LIN {X 0,Y 323.415,Z 444.934,A -85,B 0,C 180,E1 -15252.367,E2 -15252.367} C_VEL
LIN {X 0,Y 322.747,Z 443.056,A -85,B 0,C 180,E1 -15254.172,E2 -15254.172} C_VEL
LIN {X 0,Y 321.888,Z 440.789,A -85,B 0,C 180,E1 -15257.402,E2 -15257.402} C_VEL
LIN {X 0,Y 321.677,Z 439.746,A -85,B 0,C 180,E1 -15260.684,E2 -15260.684} C_VEL
LIN {X 0,Y 321.703,Z 439.751,A -85,B 0,C 180,E1 -15262.288,E2 -15262.288} C_VEL
LIN {X 0,Y 322.05,Z 441.15,A -85,B 0,C 180,E1 -15266.204,E2 -15266.204} C_VEL
LIN {X 0,Y 323.339,Z 443.035,A -85,B 0,C 180,E1 -15266.931,E2 -15266.931} C_VEL
LIN {X 0,Y 326.04,Z 445.709,A -85,B 0,C 180,E1 -15268.047,E2 -15268.047} C_VEL
LIN {X 0,Y 328.944,Z 449.026,A -85,B 0,C 180,E1 -15269.151,E2 -15269.151} C_VEL
LIN {X 0,Y 333.336,Z 454.917,A -85,B 0,C 180,E1 -15270.681,E2 -15270.681} C_VEL
LIN {X 0,Y 337.033,Z 460.145,A -85,B 0,C 180,E1 -15271.83,E2 -15271.83} C_VEL
LIN {X 0,Y 340.789,Z 466.587,A -85,B 0,C 180,E1 -15272.953,E2 -15272.953} C_VEL
LIN {X 0,Y 342.722,Z 470.945,A -85,B 0,C 180,E1 -15273.54,E2 -15273.54} C_VEL
LIN {X 0,Y 337.416,Z 532.467,A -85,B 0,C 180,E1 -15275.791,E2 -15275.791} C_VEL
LIN {X 0,Y 336.439,Z 545.574,A -85,B 0,C 180,E1 -15276.412,E2 -15276.412} C_VEL
LIN {X 0,Y 335.148,Z 559.103,A -85,B 0,C 180,E1 -15277.321,E2 -15277.321} C_VEL
LIN {X 0,Y 333.581,Z 571.352,A -85,B 0,C 180,E1 -15278.387,E2 -15278.387} C_VEL
LIN {X 0,Y 331.934,Z 581.953,A -85,B 0,C 180,E1 -15279.552,E2 -15279.552} C_VEL
LIN {X 0,Y 329.898,Z 592.789,A -85,B 0,C 180,E1 -15281.042,E2 -15281.042} C_VEL
LIN {X 0,Y 328.192,Z 601.663,A -85,B 0,C 180,E1 -15282.554,E2 -15282.554} C_VEL
LIN {X 0,Y 326.248,Z 610.311,A -85,B 0,C 180,E1 -15284.379,E2 -15284.379} C_VEL
LIN {X 0,Y 324.54,Z 617.246,A -85,B 0,C 180,E1 -15286.219,E2 -15286.219} C_VEL
LIN {X 0,Y 322.892,Z 623.517,A -85,B 0,C 180,E1 -15288.368,E2 -15288.368} C_VEL
LIN {X 0,Y 321.452,Z 628.255,A -85,B 0,C 180,E1 -15290.562,E2 -15290.562} C_VEL
LIN {X 0,Y 320.468,Z 631.089,A -85,B 0,C 180,E1 -15292.439,E2 -15292.439} C_VEL
LIN {X 0,Y 320.007,Z 632.416,A -85,B 0,C 180,E1 -15293.696,E2 -15293.696} C_VEL
LIN {X 0,Y 319.55,Z 633.281,A -85,B 0,C 180,E1 -15294.953,E2 -15294.953} C_VEL
LIN {X 0,Y 319.121,Z 633.733,A -85,B 0,C 180,E1 -15296.212,E2 -15296.212} C_VEL
LIN {X 0,Y 318.802,Z 633.773,A -85,B 0,C 180,E1 -15297.473,E2 -15297.473} C_VEL
LIN {X 0,Y 318.621,Z 633.362,A -85,B 0,C 180,E1 -15298.736,E2 -15298.736} C_VEL
LIN {X 0,Y 318.509,Z 632.498,A -85,B 0,C 180,E1 -15300,E2 -15300} C_VEL
LIN {X 0,Y 318.493,Z 631.215,A -85,B 0,C 180,E1 -15301.264,E2 -15301.264} C_VEL
LIN {X 0,Y 318.632,Z 628.449,A -85,B 0,C 180,E1 -15303.161,E2 -15303.161} C_VEL
LIN {X 0,Y 318.806,Z 624.631,A -85,B 0,C 180,E1 -15305.059,E2 -15305.059} C_VEL
LIN {X 0,Y 319.03,Z 618.858,A -85,B 0,C 180,E1 -15307.223,E2 -15307.223} C_VEL
LIN {X 0,Y 319.415,Z 612.127,A -85,B 0,C 180,E1 -15309.179,E2 -15309.179} C_VEL
LIN {X 0,Y 320.054,Z 603.989,A -85,B 0,C 180,E1 -15311.078,E2 -15311.078} C_VEL
LIN {X 0,Y 320.625,Z 595.659,A -85,B 0,C 180,E1 -15312.662,E2 -15312.662} C_VEL
LIN {X 0,Y 321.5,Z 584.421,A -85,B 0,C 180,E1 -15314.398,E2 -15314.398} C_VEL
LIN {X 0,Y 322.301,Z 572.943,A -85,B 0,C 180,E1 -15315.817,E2 -15315.817} C_VEL
LIN {X 0,Y 323.062,Z 560.1,A -85,B 0,C 180,E1 -15317.078,E2 -15317.078} C_VEL
LIN {X 0,Y 323.641,Z 547.511,A -85,B 0,C 180,E1 -15318.026,E2 -15318.026} C_VEL
LIN {X 0,Y 324.226,Z 533.31,A -85,B 0,C 180,E1 -15318.81,E2 -15318.81} C_VEL
LIN {X 0,Y 324.598,Z 516.462,A -85,B 0,C 180,E1 -15319.403,E2 -15319.403} C_VEL
LIN {X 0,Y 326.507,Z 455.246,A -85,B 0,C 180,E1 -15321.28,E2 -15321.28} C_VEL
LIN {X 0,Y 319.589,Z 433.672,A -85,B 0,C 180,E1 -15322.294,E2 -15322.294} C_VEL
LIN {X 0,Y 319.62,Z 433.67,A -85,B 0,C 180,E1 -15326.09,E2 -15326.09} C_VEL
LIN {X 0,Y 319.582,Z 433.673,A -85,B 0,C 180,E1 -15328.935,E2 -15328.935} C_VEL
LIN {X 0,Y 319.533,Z 433.672,A -85,B 0,C 180,E1 -15331.862,E2 -15331.862} C_VEL
LIN {X 0,Y 319.582,Z 433.666,A -85,B 0,C 180,E1 -15335.543,E2 -15335.543} C_VEL
LIN {X 0,Y 319.575,Z 433.679,A -85,B 0,C 180,E1 -15338.008,E2 -15338.008} C_VEL
LIN {X 0,Y 319.528,Z 433.674,A -85,B 0,C 180,E1 -15341.597,E2 -15341.597} C_VEL
LIN {X 0,Y 319.49,Z 433.675,A -85,B 0,C 180,E1 -15345.257,E2 -15345.257} C_VEL
LIN {X 0,Y 319.53,Z 433.68,A -85,B 0,C 180,E1 -15348.712,E2 -15348.712} C_VEL
LIN {X 0,Y 319.579,Z 433.675,A -85,B 0,C 180,E1 -15352.344,E2 -15352.344} C_VEL
LIN {X 0,Y 319.569,Z 433.674,A -85,B 0,C 180,E1 -15356.269,E2 -15356.269} C_VEL
LIN {X 0,Y 319.586,Z 433.759,A -85,B 0,C 180,E1 -15356.479,E2 -15356.479} C_VEL
LIN {X 0,Y 323.437,Z 448.445,A -85,B 0,C 180,E1 -15360.015,E2 -15360.015} C_VEL
LIN {X 0,Y 326.314,Z 462.259,A -85,B 0,C 180,E1 -15363.109,E2 -15363.109} C_VEL
LIN {X 0,Y 325.683,Z 473.289,A -85,B 0,C 180,E1 -15365.183,E2 -15365.183} C_VEL
LIN {X 0,Y 330.444,Z 499.684,A -85,B 0,C 180,E1 -15366.196,E2 -15366.196} C_VEL
LIN {X 0,Y 331.048,Z 503.636,A -85,B 0,C 180,E1 -15366.335,E2 -15366.335} C_VEL
LIN {X 0,Y 329.359,Z 580.024,A -85,B 0,C 180,E1 -15367.991,E2 -15367.991} C_VEL
LIN {X 0,Y 328.84,Z 592.637,A -85,B 0,C 180,E1 -15368.408,E2 -15368.408} C_VEL
LIN {X 0,Y 328.036,Z 605.004,A -85,B 0,C 180,E1 -15369.052,E2 -15369.052} C_VEL
LIN {X 0,Y 327.015,Z 616.639,A -85,B 0,C 180,E1 -15369.888,E2 -15369.888} C_VEL
LIN {X 0,Y 325.83,Z 628.009,A -85,B 0,C 180,E1 -15370.959,E2 -15370.959} C_VEL
LIN {X 0,Y 324.592,Z 638.26,A -85,B 0,C 180,E1 -15372.192,E2 -15372.192} C_VEL
LIN {X 0,Y 323.417,Z 647.66,A -85,B 0,C 180,E1 -15373.591,E2 -15373.591} C_VEL
LIN {X 0,Y 322.077,Z 656.251,A -85,B 0,C 180,E1 -15375.144,E2 -15375.144} C_VEL
LIN {X 0,Y 320.971,Z 663.34,A -85,B 0,C 180,E1 -15376.708,E2 -15376.708} C_VEL
LIN {X 0,Y 319.984,Z 670.3,A -85,B 0,C 180,E1 -15378.599,E2 -15378.599} C_VEL
LIN {X 0,Y 319.101,Z 675.831,A -85,B 0,C 180,E1 -15380.492,E2 -15380.492} C_VEL
LIN {X 0,Y 318.58,Z 680.167,A -85,B 0,C 180,E1 -15382.394,E2 -15382.394} C_VEL
LIN {X 0,Y 318.316,Z 682.449,A -85,B 0,C 180,E1 -15383.662,E2 -15383.662} C_VEL
LIN {X 0,Y 318.124,Z 684.309,A -85,B 0,C 180,E1 -15384.93,E2 -15384.93} C_VEL
LIN {X 0,Y 317.974,Z 685.729,A -85,B 0,C 180,E1 -15386.198,E2 -15386.198} C_VEL
LIN {X 0,Y 317.781,Z 687.339,A -85,B 0,C 180,E1 -15388.733,E2 -15388.733} C_VEL
LIN {X 0,Y 317.771,Z 687.572,A -85,B 0,C 180,E1 -15390,E2 -15390} C_VEL
LIN {X 0,Y 317.781,Z 687.379,A -85,B 0,C 180,E1 -15391.267,E2 -15391.267} C_VEL
LIN {X 0,Y 317.973,Z 685.821,A -85,B 0,C 180,E1 -15393.802,E2 -15393.802} C_VEL
LIN {X 0,Y 318.122,Z 684.453,A -85,B 0,C 180,E1 -15395.07,E2 -15395.07} C_VEL
LIN {X 0,Y 318.342,Z 682.27,A -85,B 0,C 180,E1 -15396.554,E2 -15396.554} C_VEL
LIN {X 0,Y 318.886,Z 677.67,A -85,B 0,C 180,E1 -15398.875,E2 -15398.875} C_VEL
LIN {X 0,Y 319.634,Z 672.603,A -85,B 0,C 180,E1 -15400.772,E2 -15400.772} C_VEL
LIN {X 0,Y 320.596,Z 666.215,A -85,B 0,C 180,E1 -15402.663,E2 -15402.663} C_VEL
LIN {X 0,Y 321.787,Z 658.275,A -85,B 0,C 180,E1 -15404.547,E2 -15404.547} C_VEL
LIN {X 0,Y 323.069,Z 650.155,A -85,B 0,C 180,E1 -15406.103,E2 -15406.103} C_VEL
LIN {X 0,Y 324.219,Z 641.396,A -85,B 0,C 180,E1 -15407.488,E2 -15407.488} C_VEL
LIN {X 0,Y 325.565,Z 630.307,A -85,B 0,C 180,E1 -15408.893,E2 -15408.893} C_VEL
LIN {X 0,Y 326.747,Z 619.606,A -85,B 0,C 180,E1 -15409.966,E2 -15409.966} C_VEL
LIN {X 0,Y 327.941,Z 607.838,A -85,B 0,C 180,E1 -15410.872,E2 -15410.872} C_VEL
LIN {X 0,Y 328.723,Z 594.884,A -85,B 0,C 180,E1 -15411.601,E2 -15411.601} C_VEL
LIN {X 0,Y 329.322,Z 582.394,A -85,B 0,C 180,E1 -15412.053,E2 -15412.053} C_VEL
LIN {X 0,Y 330.329,Z 541.842,A -85,B 0,C 180,E1 -15412.94,E2 -15412.94} C_VEL
LIN {X 0,Y 329.832,Z 536.045,A -85,B 0,C 180,E1 -15413.111,E2 -15413.111} C_VEL
LIN {X 0,Y 325.025,Z 517.382,A -85,B 0,C 180,E1 -15413.918,E2 -15413.918} C_VEL
LIN {X 0,Y 324.474,Z 511.587,A -85,B 0,C 180,E1 -15414.099,E2 -15414.099} C_VEL
LIN {X 0,Y 324.36,Z 502.656,A -85,B 0,C 180,E1 -15414.322,E2 -15414.322} C_VEL
LIN {X 0,Y 319.063,Z 473.491,A -85,B 0,C 180,E1 -15415.476,E2 -15415.476} C_VEL
LIN {X 0,Y 319.632,Z 464.637,A -85,B 0,C 180,E1 -15417.145,E2 -15417.145} C_VEL
LIN {X 0,Y 317.313,Z 452.97,A -85,B 0,C 180,E1 -15419.78,E2 -15419.78} C_VEL
LIN {X 0,Y 314.508,Z 441.94,A -85,B 0,C 180,E1 -15422.433,E2 -15422.433} C_VEL
LIN {X 0,Y 312.518,Z 434.56,A -85,B 0,C 180,E1 -15424.306,E2 -15424.306} C_VEL
LIN {X 0,Y 312.507,Z 434.556,A -85,B 0,C 180,E1 -15428.083,E2 -15428.083} C_VEL
LIN {X 0,Y 312.517,Z 434.558,A -85,B 0,C 180,E1 -15432.088,E2 -15432.088} C_VEL
LIN {X 0,Y 312.484,Z 434.564,A -85,B 0,C 180,E1 -15436.03,E2 -15436.03} C_VEL
LIN {X 0,Y 312.506,Z 434.558,A -85,B 0,C 180,E1 -15439.875,E2 -15439.875} C_VEL
LIN {X 0,Y 312.528,Z 434.542,A -85,B 0,C 180,E1 -15442.615,E2 -15442.615} C_VEL
LIN {X 0,Y 312.521,Z 434.556,A -85,B 0,C 180,E1 -15446.311,E2 -15446.311} C_VEL
LIN {X 0,Y 312.548,Z 434.584,A -85,B 0,C 180,E1 -15448.771,E2 -15448.771} C_VEL
LIN {X 0,Y 315.782,Z 449.762,A -85,B 0,C 180,E1 -15452.136,E2 -15452.136} C_VEL
LIN {X 0,Y 317.182,Z 456.988,A -85,B 0,C 180,E1 -15453.695,E2 -15453.695} C_VEL
LIN {X 0,Y 316.837,Z 466.284,A -85,B 0,C 180,E1 -15455.578,E2 -15455.578} C_VEL
LIN {X 0,Y 316.232,Z 474.416,A -85,B 0,C 180,E1 -15457.151,E2 -15457.151} C_VEL
LIN {X 0,Y 319.632,Z 503.07,A -85,B 0,C 180,E1 -15458.25,E2 -15458.25} C_VEL
LIN {X 0,Y 317.023,Z 585.287,A -85,B 0,C 180,E1 -15460.872,E2 -15460.872} C_VEL
LIN {X 0,Y 316.404,Z 598.786,A -85,B 0,C 180,E1 -15461.547,E2 -15461.547} C_VEL
LIN {X 0,Y 315.725,Z 610.437,A -85,B 0,C 180,E1 -15462.345,E2 -15462.345} C_VEL
LIN {X 0,Y 314.883,Z 623.458,A -85,B 0,C 180,E1 -15463.518,E2 -15463.518} C_VEL
LIN {X 0,Y 314.182,Z 634.377,A -85,B 0,C 180,E1 -15464.761,E2 -15464.761} C_VEL
LIN {X 0,Y 313.36,Z 644.692,A -85,B 0,C 180,E1 -15466.214,E2 -15466.214} C_VEL
LIN {X 0,Y 312.444,Z 654.963,A -85,B 0,C 180,E1 -15467.991,E2 -15467.991} C_VEL
LIN {X 0,Y 311.757,Z 663.937,A -85,B 0,C 180,E1 -15469.938,E2 -15469.938} C_VEL
LIN {X 0,Y 311.283,Z 671.121,A -85,B 0,C 180,E1 -15471.888,E2 -15471.888} C_VEL
LIN {X 0,Y 310.947,Z 677.186,A -85,B 0,C 180,E1 -15473.981,E2 -15473.981} C_VEL
LIN {X 0,Y 310.836,Z 681.89,A -85,B 0,C 180,E1 -15476.111,E2 -15476.111} C_VEL
LIN {X 0,Y 310.734,Z 684.041,A -85,B 0,C 180,E1 -15477.407,E2 -15477.407} C_VEL
LIN {X 0,Y 310.662,Z 685.752,A -85,B 0,C 180,E1 -15478.704,E2 -15478.704} C_VEL
LIN {X 0,Y 310.675,Z 687.002,A -85,B 0,C 180,E1 -15480,E2 -15480} C_VEL
LIN {X 0,Y 310.717,Z 687.784,A -85,B 0,C 180,E1 -15481.296,E2 -15481.296} C_VEL
LIN {X 0,Y 310.805,Z 688.153,A -85,B 0,C 180,E1 -15482.592,E2 -15482.592} C_VEL
LIN {X 0,Y 310.953,Z 688.067,A -85,B 0,C 180,E1 -15483.888,E2 -15483.888} C_VEL
LIN {X 0,Y 311.226,Z 687.529,A -85,B 0,C 180,E1 -15485.182,E2 -15485.182} C_VEL
LIN {X 0,Y 311.677,Z 685.878,A -85,B 0,C 180,E1 -15487.18,E2 -15487.18} C_VEL
LIN {X 0,Y 312.593,Z 682.248,A -85,B 0,C 180,E1 -15489.708,E2 -15489.708} C_VEL
LIN {X 0,Y 313.634,Z 678.194,A -85,B 0,C 180,E1 -15491.635,E2 -15491.635} C_VEL
LIN {X 0,Y 315.101,Z 672.043,A -85,B 0,C 180,E1 -15493.873,E2 -15493.873} C_VEL
LIN {X 0,Y 316.848,Z 665.229,A -85,B 0,C 180,E1 -15495.766,E2 -15495.766} C_VEL
LIN {X 0,Y 318.829,Z 656.762,A -85,B 0,C 180,E1 -15497.643,E2 -15497.643} C_VEL
LIN {X 0,Y 320.758,Z 648.266,A -85,B 0,C 180,E1 -15499.187,E2 -15499.187} C_VEL
LIN {X 0,Y 323.027,Z 637.095,A -85,B 0,C 180,E1 -15500.821,E2 -15500.821} C_VEL
LIN {X 0,Y 325.003,Z 626.38,A -85,B 0,C 180,E1 -15502.069,E2 -15502.069} C_VEL
LIN {X 0,Y 327.058,Z 613.592,A -85,B 0,C 180,E1 -15503.257,E2 -15503.257} C_VEL
LIN {X 0,Y 328.881,Z 600.055,A -85,B 0,C 180,E1 -15504.207,E2 -15504.207} C_VEL
LIN {X 0,Y 330.303,Z 587.28,A -85,B 0,C 180,E1 -15504.849,E2 -15504.849} C_VEL
LIN {X 0,Y 337.255,Z 510.337,A -85,B 0,C 180,E1 -15507.694,E2 -15507.694} C_VEL
LIN {X 0,Y 335.598,Z 498.438,A -85,B 0,C 180,E1 -15508.704,E2 -15508.704} C_VEL
LIN {X 0,Y 333.132,Z 485.763,A -85,B 0,C 180,E1 -15510.027,E2 -15510.027} C_VEL
LIN {X 0,Y 330.644,Z 480.2,A -85,B 0,C 180,E1 -15511.002,E2 -15511.002} C_VEL
LIN {X 0,Y 329.554,Z 477.674,A -85,B 0,C 180,E1 -15511.5,E2 -15511.5} C_VEL
LIN {X 0,Y 328.456,Z 471.4,A -85,B 0,C 180,E1 -15513.802,E2 -15513.802} C_VEL
LIN {X 0,Y 327.132,Z 465.762,A -85,B 0,C 180,E1 -15516.294,E2 -15516.294} C_VEL
LIN {X 0,Y 325.787,Z 461.014,A -85,B 0,C 180,E1 -15519.049,E2 -15519.049} C_VEL
LIN {X 0,Y 325,Z 458.807,A -85,B 0,C 180,E1 -15520.811,E2 -15520.811} C_VEL
LIN {X 0,Y 324.43,Z 457.206,A -85,B 0,C 180,E1 -15522.563,E2 -15522.563} C_VEL
LIN {X 0,Y 324.104,Z 456.188,A -85,B 0,C 180,E1 -15524.308,E2 -15524.308} C_VEL
LIN {X 0,Y 324.123,Z 455.716,A -85,B 0,C 180,E1 -15526.063,E2 -15526.063} C_VEL
LIN {X 0,Y 324.456,Z 455.835,A -85,B 0,C 180,E1 -15527.818,E2 -15527.818} C_VEL
LIN {X 0,Y 325.079,Z 456.625,A -85,B 0,C 180,E1 -15529.565,E2 -15529.565} C_VEL
LIN {X 0,Y 326.106,Z 457.967,A -85,B 0,C 180,E1 -15531.319,E2 -15531.319} C_VEL
LIN {X 0,Y 327.63,Z 460.057,A -85,B 0,C 180,E1 -15533.085,E2 -15533.085} C_VEL
LIN {X 0,Y 329.444,Z 463.109,A -85,B 0,C 180,E1 -15534.831,E2 -15534.831} C_VEL
LIN {X 0,Y 330.272,Z 465.705,A -85,B 0,C 180,E1 -15535.805,E2 -15535.805} C_VEL
LIN {X 0,Y 331.517,Z 476.027,A -85,B 0,C 180,E1 -15538.23,E2 -15538.23} C_VEL
LIN {X 0,Y 331.517,Z 479.248,A -85,B 0,C 180,E1 -15538.749,E2 -15538.749} C_VEL
LIN {X 0,Y 331.408,Z 483.383,A -85,B 0,C 180,E1 -15539.309,E2 -15539.309} C_VEL
LIN {X 0,Y 333.025,Z 496.79,A -85,B 0,C 180,E1 -15540.572,E2 -15540.572} C_VEL
LIN {X 0,Y 334.336,Z 512.867,A -85,B 0,C 180,E1 -15541.832,E2 -15541.832} C_VEL
LIN {X 0,Y 334.671,Z 523.859,A -85,B 0,C 180,E1 -15542.527,E2 -15542.527} C_VEL
LIN {X 0,Y 334.534,Z 534.014,A -85,B 0,C 180,E1 -15543.081,E2 -15543.081} C_VEL
LIN {X 0,Y 327.846,Z 607.437,A -85,B 0,C 180,E1 -15545.88,E2 -15545.88} C_VEL
LIN {X 0,Y 326.268,Z 620.214,A -85,B 0,C 180,E1 -15546.6,E2 -15546.6} C_VEL
LIN {X 0,Y 324.344,Z 632.764,A -85,B 0,C 180,E1 -15547.548,E2 -15547.548} C_VEL
LIN {X 0,Y 322.229,Z 644.83,A -85,B 0,C 180,E1 -15548.74,E2 -15548.74} C_VEL
LIN {X 0,Y 320.177,Z 655.866,A -85,B 0,C 180,E1 -15550.109,E2 -15550.109} C_VEL
LIN {X 0,Y 318.179,Z 665.815,A -85,B 0,C 180,E1 -15551.654,E2 -15551.654} C_VEL
LIN {X 0,Y 316.075,Z 675.567,A -85,B 0,C 180,E1 -15553.531,E2 -15553.531} C_VEL
LIN {X 0,Y 314.407,Z 683.427,A -85,B 0,C 180,E1 -15555.435,E2 -15555.435} C_VEL
LIN {X 0,Y 313.303,Z 688.803,A -85,B 0,C 180,E1 -15557.037,E2 -15557.037} C_VEL
LIN {X 0,Y 312.222,Z 694.016,A -85,B 0,C 180,E1 -15558.969,E2 -15558.969} C_VEL
LIN {X 0,Y 311.496,Z 698.068,A -85,B 0,C 180,E1 -15560.913,E2 -15560.913} C_VEL
LIN {X 0,Y 311.174,Z 700.166,A -85,B 0,C 180,E1 -15562.212,E2 -15562.212} C_VEL
LIN {X 0,Y 310.841,Z 702.425,A -85,B 0,C 180,E1 -15564.169,E2 -15564.169} C_VEL
LIN {X 0,Y 310.773,Z 703.655,A -85,B 0,C 180,E1 -15566.11,E2 -15566.11} C_VEL
LIN {X 0,Y 310.756,Z 704.314,A -85,B 0,C 180,E1 -15570,E2 -15570} C_VEL
LIN {X 0,Y 310.707,Z 704.088,A -85,B 0,C 180,E1 -15571.296,E2 -15571.296} C_VEL
LIN {X 0,Y 310.734,Z 703.469,A -85,B 0,C 180,E1 -15572.593,E2 -15572.593} C_VEL
LIN {X 0,Y 310.768,Z 702.458,A -85,B 0,C 180,E1 -15573.89,E2 -15573.89} C_VEL
LIN {X 0,Y 310.795,Z 700.254,A -85,B 0,C 180,E1 -15575.746,E2 -15575.746} C_VEL
LIN {X 0,Y 311.048,Z 696.794,A -85,B 0,C 180,E1 -15577.791,E2 -15577.791} C_VEL
LIN {X 0,Y 311.501,Z 692.373,A -85,B 0,C 180,E1 -15579.742,E2 -15579.742} C_VEL
LIN {X 0,Y 312.159,Z 686.737,A -85,B 0,C 180,E1 -15581.691,E2 -15581.691} C_VEL
LIN {X 0,Y 313.226,Z 679.645,A -85,B 0,C 180,E1 -15583.627,E2 -15583.627} C_VEL
LIN {X 0,Y 314.513,Z 670.786,A -85,B 0,C 180,E1 -15585.554,E2 -15585.554} C_VEL
LIN {X 0,Y 315.78,Z 661.681,A -85,B 0,C 180,E1 -15587.151,E2 -15587.151} C_VEL
LIN {X 0,Y 317.15,Z 651.544,A -85,B 0,C 180,E1 -15588.575,E2 -15588.575} C_VEL
LIN {X 0,Y 317.887,Z 646.645,A -85,B 0,C 180,E1 -15589.2,E2 -15589.2} C_VEL
LIN {X 0,Y 320.208,Z 636.026,A -85,B 0,C 180,E1 -15590.727,E2 -15590.727} C_VEL
LIN {X 0,Y 322.584,Z 624.425,A -85,B 0,C 180,E1 -15592.075,E2 -15592.075} C_VEL
LIN {X 0,Y 324.719,Z 613.46,A -85,B 0,C 180,E1 -15593.097,E2 -15593.097} C_VEL
LIN {X 0,Y 327.191,Z 598.598,A -85,B 0,C 180,E1 -15594.171,E2 -15594.171} C_VEL
LIN {X 0,Y 329.121,Z 584.613,A -85,B 0,C 180,E1 -15594.902,E2 -15594.902} C_VEL
LIN {X 0,Y 333.639,Z 531.163,A -85,B 0,C 180,E1 -15596.899,E2 -15596.899} C_VEL
LIN {X 0,Y 333.322,Z 518.201,A -85,B 0,C 180,E1 -15597.637,E2 -15597.637} C_VEL
LIN {X 0,Y 332.158,Z 504.388,A -85,B 0,C 180,E1 -15598.615,E2 -15598.615} C_VEL
LIN {X 0,Y 330.494,Z 491.797,A -85,B 0,C 180,E1 -15599.692,E2 -15599.692} C_VEL
LIN {X 0,Y 328.256,Z 478.757,A -85,B 0,C 180,E1 -15601.02,E2 -15601.02} C_VEL
LIN {X 0,Y 327.534,Z 476.371,A -85,B 0,C 180,E1 -15601.358,E2 -15601.358} C_VEL
LIN {X 0,Y 324.779,Z 470.229,A -85,B 0,C 180,E1 -15602.501,E2 -15602.501} C_VEL
LIN {X 0,Y 321.451,Z 463.195,A -85,B 0,C 180,E1 -15604.058,E2 -15604.058} C_VEL
LIN {X 0,Y 320.307,Z 458.211,A -85,B 0,C 180,E1 -15606.329,E2 -15606.329} C_VEL
LIN {X 0,Y 318.674,Z 452.607,A -85,B 0,C 180,E1 -15609.476,E2 -15609.476} C_VEL
LIN {X 0,Y 317.754,Z 449.671,A -85,B 0,C 180,E1 -15611.57,E2 -15611.57} C_VEL
LIN {X 0,Y 316.573,Z 446.395,A -85,B 0,C 180,E1 -15614.732,E2 -15614.732} C_VEL
LIN {X 0,Y 315.819,Z 444.294,A -85,B 0,C 180,E1 -15618.118,E2 -15618.118} C_VEL
LIN {X 0,Y 315.693,Z 443.542,A -85,B 0,C 180,E1 -15621.185,E2 -15621.185} C_VEL
LIN {X 0,Y 315.715,Z 443.892,A -85,B 0,C 180,E1 -15623.809,E2 -15623.809} C_VEL
LIN {X 0,Y 318.034,Z 446.624,A -85,B 0,C 180,E1 -15625.246,E2 -15625.246} C_VEL
LIN {X 0,Y 319.827,Z 448.076,A -85,B 0,C 180,E1 -15626.133,E2 -15626.133} C_VEL
LIN {X 0,Y 322.66,Z 451.25,A -85,B 0,C 180,E1 -15627.448,E2 -15627.448} C_VEL
LIN {X 0,Y 326.879,Z 456.492,A -85,B 0,C 180,E1 -15629.15,E2 -15629.15} C_VEL
LIN {X 0,Y 331.321,Z 462.561,A -85,B 0,C 180,E1 -15630.72,E2 -15630.72} C_VEL
LIN {X 0,Y 335.075,Z 468.45,A -85,B 0,C 180,E1 -15631.927,E2 -15631.927} C_VEL
LIN {X 0,Y 337.55,Z 473.445,A -85,B 0,C 180,E1 -15632.738,E2 -15632.738} C_VEL
LIN {X 0,Y 332.009,Z 533.902,A -85,B 0,C 180,E1 -15635.037,E2 -15635.037} C_VEL
LIN {X 0,Y 330.972,Z 546.82,A -85,B 0,C 180,E1 -15635.664,E2 -15635.664} C_VEL
LIN {X 0,Y 329.588,Z 560.2,A -85,B 0,C 180,E1 -15636.583,E2 -15636.583} C_VEL
LIN {X 0,Y 327.696,Z 573.546,A -85,B 0,C 180,E1 -15637.795,E2 -15637.795} C_VEL
LIN {X 0,Y 325.451,Z 586.247,A -85,B 0,C 180,E1 -15639.292,E2 -15639.292} C_VEL
LIN {X 0,Y 323.574,Z 595.55,A -85,B 0,C 180,E1 -15640.657,E2 -15640.657} C_VEL
LIN {X 0,Y 321.374,Z 605.509,A -85,B 0,C 180,E1 -15642.501,E2 -15642.501} C_VEL
LIN {X 0,Y 319.361,Z 613.545,A -85,B 0,C 180,E1 -15644.361,E2 -15644.361} C_VEL
LIN {X 0,Y 317.869,Z 619.049,A -85,B 0,C 180,E1 -15645.924,E2 -15645.924} C_VEL
LIN {X 0,Y 316.285,Z 624.492,A -85,B 0,C 180,E1 -15647.879,E2 -15647.879} C_VEL
LIN {X 0,Y 314.961,Z 628.444,A -85,B 0,C 180,E1 -15649.717,E2 -15649.717} C_VEL
LIN {X 0,Y 314.142,Z 630.572,A -85,B 0,C 180,E1 -15650.99,E2 -15650.99} C_VEL
LIN {X 0,Y 313.527,Z 632.26,A -85,B 0,C 180,E1 -15652.271,E2 -15652.271} C_VEL
LIN {X 0,Y 313.027,Z 633.461,A -85,B 0,C 180,E1 -15653.554,E2 -15653.554} C_VEL
LIN {X 0,Y 312.545,Z 634.237,A -85,B 0,C 180,E1 -15654.84,E2 -15654.84} C_VEL
LIN {X 0,Y 312.1,Z 634.605,A -85,B 0,C 180,E1 -15656.126,E2 -15656.126} C_VEL
LIN {X 0,Y 311.769,Z 634.539,A -85,B 0,C 180,E1 -15657.416,E2 -15657.416} C_VEL
LIN {X 0,Y 311.581,Z 634.003,A -85,B 0,C 180,E1 -15658.708,E2 -15658.708} C_VEL
LIN {X 0,Y 311.436,Z 633.063,A -85,B 0,C 180,E1 -15660,E2 -15660} C_VEL
LIN {X 0,Y 311.426,Z 631.699,A -85,B 0,C 180,E1 -15661.293,E2 -15661.293} C_VEL
LIN {X 0,Y 311.574,Z 628.777,A -85,B 0,C 180,E1 -15663.233,E2 -15663.233} C_VEL
LIN {X 0,Y 311.734,Z 624.786,A -85,B 0,C 180,E1 -15665.174,E2 -15665.174} C_VEL
LIN {X 0,Y 311.935,Z 619.311,A -85,B 0,C 180,E1 -15667.212,E2 -15667.212} C_VEL
LIN {X 0,Y 312.378,Z 611.845,A -85,B 0,C 180,E1 -15669.388,E2 -15669.388} C_VEL
LIN {X 0,Y 313.034,Z 603.434,A -85,B 0,C 180,E1 -15671.329,E2 -15671.329} C_VEL
LIN {X 0,Y 313.814,Z 592.981,A -85,B 0,C 180,E1 -15673.271,E2 -15673.271} C_VEL
LIN {X 0,Y 314.649,Z 582.091,A -85,B 0,C 180,E1 -15674.884,E2 -15674.884} C_VEL
LIN {X 0,Y 315.387,Z 571.39,A -85,B 0,C 180,E1 -15676.174,E2 -15676.174} C_VEL
LIN {X 0,Y 316.049,Z 560.346,A -85,B 0,C 180,E1 -15677.253,E2 -15677.253} C_VEL
LIN {X 0,Y 316.676,Z 546.889,A -85,B 0,C 180,E1 -15678.269,E2 -15678.269} C_VEL
LIN {X 0,Y 317.225,Z 532.968,A -85,B 0,C 180,E1 -15679.032,E2 -15679.032} C_VEL
LIN {X 0,Y 317.697,Z 513.307,A -85,B 0,C 180,E1 -15679.716,E2 -15679.716} C_VEL
LIN {X 0,Y 319.433,Z 456.164,A -85,B 0,C 180,E1 -15681.526,E2 -15681.526} C_VEL
LIN {X 0,Y 312.562,Z 434.547,A -85,B 0,C 180,E1 -15682.571,E2 -15682.571} C_VEL
LIN {X 0,Y 312.599,Z 434.545,A -85,B 0,C 180,E1 -15685.933,E2 -15685.933} C_VEL
LIN {X 0,Y 312.54,Z 434.554,A -85,B 0,C 180,E1 -15689.651,E2 -15689.651} C_VEL
LIN {X 0,Y 312.521,Z 434.528,A -85,B 0,C 180,E1 -15693.689,E2 -15693.689} C_VEL
LIN {X 0,Y 312.528,Z 434.559,A -85,B 0,C 180,E1 -15697.385,E2 -15697.385} C_VEL
LIN {X 0,Y 312.492,Z 434.542,A -85,B 0,C 180,E1 -15700.709,E2 -15700.709} C_VEL
LIN {X 0,Y 312.454,Z 434.565,A -85,B 0,C 180,E1 -15704.21,E2 -15704.21} C_VEL
LIN {X 0,Y 312.486,Z 434.561,A -85,B 0,C 180,E1 -15707.919,E2 -15707.919} C_VEL
LIN {X 0,Y 312.536,Z 434.556,A -85,B 0,C 180,E1 -15711.911,E2 -15711.911} C_VEL
LIN {X 0,Y 312.541,Z 434.604,A -85,B 0,C 180,E1 -15715.873,E2 -15715.873} C_VEL
LIN {X 0,Y 316.178,Z 448.314,A -85,B 0,C 180,E1 -15719.253,E2 -15719.253} C_VEL
LIN {X 0,Y 318.728,Z 459.655,A -85,B 0,C 180,E1 -15721.886,E2 -15721.886} C_VEL
LIN {X 0,Y 319.585,Z 464.036,A -85,B 0,C 180,E1 -15722.85,E2 -15722.85} C_VEL
LIN {X 0,Y 319.075,Z 473.504,A -85,B 0,C 180,E1 -15724.644,E2 -15724.644} C_VEL
LIN {X 0,Y 324.308,Z 502.768,A -85,B 0,C 180,E1 -15725.789,E2 -15725.789} C_VEL
LIN {X 0,Y 324.481,Z 506.884,A -85,B 0,C 180,E1 -15725.901,E2 -15725.901} C_VEL
LIN {X 0,Y 322.812,Z 580.135,A -85,B 0,C 180,E1 -15727.52,E2 -15727.52} C_VEL
LIN {X 0,Y 322.264,Z 592.79,A -85,B 0,C 180,E1 -15727.944,E2 -15727.944} C_VEL
LIN {X 0,Y 321.32,Z 606.395,A -85,B 0,C 180,E1 -15728.677,E2 -15728.677} C_VEL
LIN {X 0,Y 320.152,Z 618.646,A -85,B 0,C 180,E1 -15729.605,E2 -15729.605} C_VEL
LIN {X 0,Y 318.771,Z 630.94,A -85,B 0,C 180,E1 -15730.855,E2 -15730.855} C_VEL
LIN {X 0,Y 317.532,Z 640.786,A -85,B 0,C 180,E1 -15732.126,E2 -15732.126} C_VEL
LIN {X 0,Y 316.338,Z 649.736,A -85,B 0,C 180,E1 -15733.545,E2 -15733.545} C_VEL
LIN {X 0,Y 314.689,Z 659.426,A -85,B 0,C 180,E1 -15735.449,E2 -15735.449} C_VEL
LIN {X 0,Y 313.524,Z 667.206,A -85,B 0,C 180,E1 -15737.376,E2 -15737.376} C_VEL
LIN {X 0,Y 312.706,Z 672.461,A -85,B 0,C 180,E1 -15738.987,E2 -15738.987} C_VEL
LIN {X 0,Y 311.865,Z 677.597,A -85,B 0,C 180,E1 -15740.924,E2 -15740.924} C_VEL
LIN {X 0,Y 311.384,Z 681.57,A -85,B 0,C 180,E1 -15742.87,E2 -15742.87} C_VEL
LIN {X 0,Y 311.059,Z 684.498,A -85,B 0,C 180,E1 -15744.815,E2 -15744.815} C_VEL
LIN {X 0,Y 310.911,Z 685.918,A -85,B 0,C 180,E1 -15746.112,E2 -15746.112} C_VEL
LIN {X 0,Y 310.695,Z 687.528,A -85,B 0,C 180,E1 -15748.704,E2 -15748.704} C_VEL
LIN {X 0,Y 310.682,Z 687.761,A -85,B 0,C 180,E1 -15750,E2 -15750} C_VEL
LIN {X 0,Y 310.695,Z 687.567,A -85,B 0,C 180,E1 -15751.296,E2 -15751.296} C_VEL
LIN {X 0,Y 310.91,Z 686.009,A -85,B 0,C 180,E1 -15753.888,E2 -15753.888} C_VEL
LIN {X 0,Y 311.057,Z 684.641,A -85,B 0,C 180,E1 -15755.185,E2 -15755.185} C_VEL
LIN {X 0,Y 311.375,Z 681.766,A -85,B 0,C 180,E1 -15757.13,E2 -15757.13} C_VEL
LIN {X 0,Y 311.863,Z 677.857,A -85,B 0,C 180,E1 -15759.076,E2 -15759.076} C_VEL
LIN {X 0,Y 312.641,Z 672.789,A -85,B 0,C 180,E1 -15761.016,E2 -15761.016} C_VEL
LIN {X 0,Y 313.654,Z 666.399,A -85,B 0,C 180,E1 -15762.948,E2 -15762.948} C_VEL
LIN {X 0,Y 314.934,Z 658.457,A -85,B 0,C 180,E1 -15764.87,E2 -15764.87} C_VEL
LIN {X 0,Y 316.259,Z 650.335,A -85,B 0,C 180,E1 -15766.459,E2 -15766.459} C_VEL
LIN {X 0,Y 317.584,Z 640.342,A -85,B 0,C 180,E1 -15768.048,E2 -15768.048} C_VEL
LIN {X 0,Y 319.077,Z 629.101,A -85,B 0,C 180,E1 -15769.46,E2 -15769.46} C_VEL
LIN {X 0,Y 320.286,Z 618.06,A -85,B 0,C 180,E1 -15770.554,E2 -15770.554} C_VEL
LIN {X 0,Y 321.467,Z 605.569,A -85,B 0,C 180,E1 -15771.481,E2 -15771.481} C_VEL
LIN {X 0,Y 322.26,Z 592.492,A -85,B 0,C 180,E1 -15772.183,E2 -15772.183} C_VEL
LIN {X 0,Y 322.864,Z 579.525,A -85,B 0,C 180,E1 -15772.603,E2 -15772.603} C_VEL
LIN {X 0,Y 324.474,Z 511.587,A -85,B 0,C 180,E1 -15774.099,E2 -15774.099} C_VEL
LIN {X 0,Y 323.77,Z 507.814,A -85,B 0,C 180,E1 -15774.245,E2 -15774.245} C_VEL
LIN {X 0,Y 320.739,Z 502.251,A -85,B 0,C 180,E1 -15774.625,E2 -15774.625} C_VEL
LIN {X 0,Y 317.344,Z 496.767,A -85,B 0,C 180,E1 -15775.041,E2 -15775.041} C_VEL
LIN {X 0,Y 316.099,Z 493.068,A -85,B 0,C 180,E1 -15775.239,E2 -15775.239} C_VEL
LIN {X 0,Y 312.438,Z 473.453,A -85,B 0,C 180,E1 -15776.083,E2 -15776.083} C_VEL
LIN {X 0,Y 312.915,Z 466.471,A -85,B 0,C 180,E1 -15777.415,E2 -15777.415} C_VEL
LIN {X 0,Y 310.499,Z 454.447,A -85,B 0,C 180,E1 -15780.175,E2 -15780.175} C_VEL
LIN {X 0,Y 307.856,Z 444.155,A -85,B 0,C 180,E1 -15782.675,E2 -15782.675} C_VEL
LIN {X 0,Y 305.483,Z 435.434,A -85,B 0,C 180,E1 -15784.903,E2 -15784.903} C_VEL
LIN {X 0,Y 305.451,Z 435.437,A -85,B 0,C 180,E1 -15788.529,E2 -15788.529} C_VEL
LIN {X 0,Y 305.479,Z 435.433,A -85,B 0,C 180,E1 -15792.59,E2 -15792.59} C_VEL
LIN {X 0,Y 305.445,Z 435.442,A -85,B 0,C 180,E1 -15796.348,E2 -15796.348} C_VEL
LIN {X 0,Y 305.46,Z 435.435,A -85,B 0,C 180,E1 -15799.892,E2 -15799.892} C_VEL
LIN {X 0,Y 305.483,Z 435.413,A -85,B 0,C 180,E1 -15803.631,E2 -15803.631} C_VEL
LIN {X 0,Y 305.468,Z 435.436,A -85,B 0,C 180,E1 -15806.483,E2 -15806.483} C_VEL
LIN {X 0,Y 305.516,Z 435.507,A -85,B 0,C 180,E1 -15808.514,E2 -15808.514} C_VEL
LIN {X 0,Y 308.85,Z 451.198,A -85,B 0,C 180,E1 -15812.025,E2 -15812.025} C_VEL
LIN {X 0,Y 310.275,Z 459.229,A -85,B 0,C 180,E1 -15813.788,E2 -15813.788} C_VEL
LIN {X 0,Y 309.486,Z 471.23,A -85,B 0,C 180,E1 -15816.229,E2 -15816.229} C_VEL
LIN {X 0,Y 309.261,Z 474.201,A -85,B 0,C 180,E1 -15816.832,E2 -15816.832} C_VEL
LIN {X 0,Y 312.42,Z 500.64,A -85,B 0,C 180,E1 -15817.883,E2 -15817.883} C_VEL
LIN {X 0,Y 312.667,Z 504.362,A -85,B 0,C 180,E1 -15818.02,E2 -15818.02} C_VEL
LIN {X 0,Y 309.967,Z 586.226,A -85,B 0,C 180,E1 -15820.72,E2 -15820.72} C_VEL
LIN {X 0,Y 309.371,Z 600.187,A -85,B 0,C 180,E1 -15821.455,E2 -15821.455} C_VEL
LIN {X 0,Y 308.477,Z 613.341,A -85,B 0,C 180,E1 -15822.43,E2 -15822.43} C_VEL
LIN {X 0,Y 307.706,Z 624.914,A -85,B 0,C 180,E1 -15823.539,E2 -15823.539} C_VEL
LIN {X 0,Y 306.948,Z 636.2,A -85,B 0,C 180,E1 -15824.903,E2 -15824.903} C_VEL
LIN {X 0,Y 306.116,Z 646.236,A -85,B 0,C 180,E1 -15826.389,E2 -15826.389} C_VEL
LIN {X 0,Y 305.301,Z 655.382,A -85,B 0,C 180,E1 -15828.043,E2 -15828.043} C_VEL
LIN {X 0,Y 304.634,Z 664.321,A -85,B 0,C 180,E1 -15830.036,E2 -15830.036} C_VEL
LIN {X 0,Y 304.154,Z 671.473,A -85,B 0,C 180,E1 -15832.031,E2 -15832.031} C_VEL
LIN {X 0,Y 303.84,Z 677.227,A -85,B 0,C 180,E1 -15834.054,E2 -15834.054} C_VEL
LIN {X 0,Y 303.753,Z 681.571,A -85,B 0,C 180,E1 -15836.02,E2 -15836.02} C_VEL
LIN {X 0,Y 303.663,Z 683.868,A -85,B 0,C 180,E1 -15837.347,E2 -15837.347} C_VEL
LIN {X 0,Y 303.58,Z 685.654,A -85,B 0,C 180,E1 -15838.673,E2 -15838.673} C_VEL
LIN {X 0,Y 303.588,Z 687.007,A -85,B 0,C 180,E1 -15840,E2 -15840} C_VEL
LIN {X 0,Y 303.633,Z 687.889,A -85,B 0,C 180,E1 -15841.326,E2 -15841.326} C_VEL
LIN {X 0,Y 303.73,Z 688.329,A -85,B 0,C 180,E1 -15842.652,E2 -15842.652} C_VEL
LIN {X 0,Y 303.896,Z 688.36,A -85,B 0,C 180,E1 -15843.978,E2 -15843.978} C_VEL
LIN {X 0,Y 304.165,Z 687.929,A -85,B 0,C 180,E1 -15845.303,E2 -15845.303} C_VEL
LIN {X 0,Y 304.616,Z 686.557,A -85,B 0,C 180,E1 -15847.213,E2 -15847.213} C_VEL
LIN {X 0,Y 305.654,Z 683.007,A -85,B 0,C 180,E1 -15849.93,E2 -15849.93} C_VEL
LIN {X 0,Y 306.746,Z 679.172,A -85,B 0,C 180,E1 -15851.9,E2 -15851.9} C_VEL
LIN {X 0,Y 308.047,Z 674.16,A -85,B 0,C 180,E1 -15853.86,E2 -15853.86} C_VEL
LIN {X 0,Y 310.174,Z 666.641,A -85,B 0,C 180,E1 -15856.115,E2 -15856.115} C_VEL
LIN {X 0,Y 312.266,Z 658.544,A -85,B 0,C 180,E1 -15858.027,E2 -15858.027} C_VEL
LIN {X 0,Y 314.732,Z 648.478,A -85,B 0,C 180,E1 -15859.91,E2 -15859.91} C_VEL
LIN {X 0,Y 317.25,Z 637.019,A -85,B 0,C 180,E1 -15861.61,E2 -15861.61} C_VEL
LIN {X 0,Y 319.557,Z 625.354,A -85,B 0,C 180,E1 -15862.978,E2 -15862.978} C_VEL
LIN {X 0,Y 321.484,Z 614.107,A -85,B 0,C 180,E1 -15864.027,E2 -15864.027} C_VEL
LIN {X 0,Y 323.392,Z 600.689,A -85,B 0,C 180,E1 -15864.987,E2 -15864.987} C_VEL
LIN {X 0,Y 324.973,Z 587.602,A -85,B 0,C 180,E1 -15865.671,E2 -15865.671} C_VEL
LIN {X 0,Y 332.402,Z 512.018,A -85,B 0,C 180,E1 -15868.553,E2 -15868.553} C_VEL
LIN {X 0,Y 330.988,Z 501.166,A -85,B 0,C 180,E1 -15869.515,E2 -15869.515} C_VEL
LIN {X 0,Y 328.988,Z 489.845,A -85,B 0,C 180,E1 -15870.748,E2 -15870.748} C_VEL
LIN {X 0,Y 325.93,Z 482.815,A -85,B 0,C 180,E1 -15872.083,E2 -15872.083} C_VEL
LIN {X 0,Y 323.627,Z 478.075,A -85,B 0,C 180,E1 -15873.218,E2 -15873.218} C_VEL
LIN {X 0,Y 322.374,Z 471.567,A -85,B 0,C 180,E1 -15876.059,E2 -15876.059} C_VEL
LIN {X 0,Y 321.519,Z 467.9,A -85,B 0,C 180,E1 -15878.102,E2 -15878.102} C_VEL
LIN {X 0,Y 320.775,Z 465.359,A -85,B 0,C 180,E1 -15879.93,E2 -15879.93} C_VEL
LIN {X 0,Y 320.225,Z 463.494,A -85,B 0,C 180,E1 -15881.737,E2 -15881.737} C_VEL
LIN {X 0,Y 319.835,Z 461.739,A -85,B 0,C 180,E1 -15884.681,E2 -15884.681} C_VEL
LIN {X 0,Y 320.115,Z 461.482,A -85,B 0,C 180,E1 -15887.11,E2 -15887.11} C_VEL
LIN {X 0,Y 320.722,Z 462.102,A -85,B 0,C 180,E1 -15888.899,E2 -15888.899} C_VEL
LIN {X 0,Y 322.471,Z 464.255,A -85,B 0,C 180,E1 -15891.683,E2 -15891.683} C_VEL
LIN {X 0,Y 323.222,Z 465.117,A -85,B 0,C 180,E1 -15892.496,E2 -15892.496} C_VEL
LIN {X 0,Y 324.865,Z 468.078,A -85,B 0,C 180,E1 -15894.26,E2 -15894.26} C_VEL
LIN {X 0,Y 325.728,Z 469.837,A -85,B 0,C 180,E1 -15895.075,E2 -15895.075} C_VEL
LIN {X 0,Y 326.202,Z 474.378,A -85,B 0,C 180,E1 -15896.29,E2 -15896.29} C_VEL
LIN {X 0,Y 326.899,Z 481.186,A -85,B 0,C 180,E1 -15897.82,E2 -15897.82} C_VEL
LIN {X 0,Y 326.957,Z 483.959,A -85,B 0,C 180,E1 -15898.189,E2 -15898.189} C_VEL
LIN {X 0,Y 328.383,Z 497.39,A -85,B 0,C 180,E1 -15899.542,E2 -15899.542} C_VEL
LIN {X 0,Y 329.447,Z 510.97,A -85,B 0,C 180,E1 -15900.69,E2 -15900.69} C_VEL
LIN {X 0,Y 329.811,Z 523.989,A -85,B 0,C 180,E1 -15901.595,E2 -15901.595} C_VEL
LIN {X 0,Y 329.601,Z 535.195,A -85,B 0,C 180,E1 -15902.224,E2 -15902.224} C_VEL
LIN {X 0,Y 322.529,Z 606.702,A -85,B 0,C 180,E1 -15905.027,E2 -15905.027} C_VEL
LIN {X 0,Y 320.831,Z 619.388,A -85,B 0,C 180,E1 -15905.749,E2 -15905.749} C_VEL
LIN {X 0,Y 318.632,Z 632.767,A -85,B 0,C 180,E1 -15906.78,E2 -15906.78} C_VEL
LIN {X 0,Y 316.377,Z 644.778,A -85,B 0,C 180,E1 -15907.984,E2 -15907.984} C_VEL
LIN {X 0,Y 314.147,Z 655.659,A -85,B 0,C 180,E1 -15909.369,E2 -15909.369} C_VEL
LIN {X 0,Y 311.906,Z 665.891,A -85,B 0,C 180,E1 -15910.998,E2 -15910.998} C_VEL
LIN {X 0,Y 309.714,Z 675.301,A -85,B 0,C 180,E1 -15912.843,E2 -15912.843} C_VEL
LIN {X 0,Y 307.867,Z 683.102,A -85,B 0,C 180,E1 -15914.78,E2 -15914.78} C_VEL
LIN {X 0,Y 306.425,Z 689.432,A -85,B 0,C 180,E1 -15916.741,E2 -15916.741} C_VEL
LIN {X 0,Y 305.268,Z 694.477,A -85,B 0,C 180,E1 -15918.715,E2 -15918.715} C_VEL
LIN {X 0,Y 304.47,Z 698.336,A -85,B 0,C 180,E1 -15920.701,E2 -15920.701} C_VEL
LIN {X 0,Y 304.109,Z 700.316,A -85,B 0,C 180,E1 -15922.03,E2 -15922.03} C_VEL
LIN {X 0,Y 303.735,Z 702.583,A -85,B 0,C 180,E1 -15924.247,E2 -15924.247} C_VEL
LIN {X 0,Y 303.687,Z 703.527,A -85,B 0,C 180,E1 -15926.019,E2 -15926.019} C_VEL
LIN {X 0,Y 303.665,Z 704.125,A -85,B 0,C 180,E1 -15930,E2 -15930} C_VEL
LIN {X 0,Y 303.622,Z 703.899,A -85,B 0,C 180,E1 -15931.326,E2 -15931.326} C_VEL
LIN {X 0,Y 303.657,Z 703.28,A -85,B 0,C 180,E1 -15932.653,E2 -15932.653} C_VEL
LIN {X 0,Y 303.68,Z 702.269,A -85,B 0,C 180,E1 -15933.981,E2 -15933.981} C_VEL
LIN {X 0,Y 303.691,Z 700.347,A -85,B 0,C 180,E1 -15935.671,E2 -15935.671} C_VEL
LIN {X 0,Y 304.005,Z 696.605,A -85,B 0,C 180,E1 -15937.973,E2 -15937.973} C_VEL
LIN {X 0,Y 304.461,Z 692.183,A -85,B 0,C 180,E1 -15939.97,E2 -15939.97} C_VEL
LIN {X 0,Y 305.168,Z 686.548,A -85,B 0,C 180,E1 -15941.962,E2 -15941.962} C_VEL
LIN {X 0,Y 306.302,Z 679.457,A -85,B 0,C 180,E1 -15943.941,E2 -15943.941} C_VEL
LIN {X 0,Y 307.674,Z 670.6,A -85,B 0,C 180,E1 -15945.909,E2 -15945.909} C_VEL
LIN {X 0,Y 308.951,Z 661.496,A -85,B 0,C 180,E1 -15947.542,E2 -15947.542} C_VEL
LIN {X 0,Y 310.614,Z 650.294,A -85,B 0,C 180,E1 -15949.152,E2 -15949.152} C_VEL
LIN {X 0,Y 313.12,Z 639.603,A -85,B 0,C 180,E1 -15950.874,E2 -15950.874} C_VEL
LIN {X 0,Y 315.835,Z 627.711,A -85,B 0,C 180,E1 -15952.4,E2 -15952.4} C_VEL
LIN {X 0,Y 318.327,Z 616.089,A -85,B 0,C 180,E1 -15953.588,E2 -15953.588} C_VEL
LIN {X 0,Y 321.062,Z 601.462,A -85,B 0,C 180,E1 -15954.749,E2 -15954.749} C_VEL
LIN {X 0,Y 323.439,Z 586.088,A -85,B 0,C 180,E1 -15955.629,E2 -15955.629} C_VEL
LIN {X 0,Y 325.049,Z 570.669,A -85,B 0,C 180,E1 -15956.268,E2 -15956.268} C_VEL
LIN {X 0,Y 328.495,Z 531.382,A -85,B 0,C 180,E1 -15957.77,E2 -15957.77} C_VEL
LIN {X 0,Y 328.293,Z 519.501,A -85,B 0,C 180,E1 -15958.481,E2 -15958.481} C_VEL
LIN {X 0,Y 327.226,Z 505.279,A -85,B 0,C 180,E1 -15959.543,E2 -15959.543} C_VEL
LIN {X 0,Y 325.71,Z 493.225,A -85,B 0,C 180,E1 -15960.648,E2 -15960.648} C_VEL
LIN {X 0,Y 323.921,Z 481.688,A -85,B 0,C 180,E1 -15961.882,E2 -15961.882} C_VEL
LIN {X 0,Y 321.209,Z 475.38,A -85,B 0,C 180,E1 -15963.107,E2 -15963.107} C_VEL
LIN {X 0,Y 317.854,Z 468.239,A -85,B 0,C 180,E1 -15964.781,E2 -15964.781} C_VEL
LIN {X 0,Y 313.621,Z 459.913,A -85,B 0,C 180,E1 -15967.354,E2 -15967.354} C_VEL
LIN {X 0,Y 312.358,Z 455.467,A -85,B 0,C 180,E1 -15970.093,E2 -15970.093} C_VEL
LIN {X 0,Y 311.29,Z 452.259,A -85,B 0,C 180,E1 -15972.634,E2 -15972.634} C_VEL
LIN {X 0,Y 310.432,Z 449.708,A -85,B 0,C 180,E1 -15975.426,E2 -15975.426} C_VEL
LIN {X 0,Y 309.806,Z 447.868,A -85,B 0,C 180,E1 -15978.862,E2 -15978.862} C_VEL
LIN {X 0,Y 309.808,Z 447.619,A -85,B 0,C 180,E1 -15980.377,E2 -15980.377} C_VEL
LIN {X 0,Y 312.772,Z 450.203,A -85,B 0,C 180,E1 -15983.075,E2 -15983.075} C_VEL
LIN {X 0,Y 313.764,Z 450.947,A -85,B 0,C 180,E1 -15983.743,E2 -15983.743} C_VEL
LIN {X 0,Y 316.472,Z 453.801,A -85,B 0,C 180,E1 -15985.387,E2 -15985.387} C_VEL
LIN {X 0,Y 317.584,Z 454.942,A -85,B 0,C 180,E1 -15985.967,E2 -15985.967} C_VEL
LIN {X 0,Y 320.683,Z 458.544,A -85,B 0,C 180,E1 -15987.451,E2 -15987.451} C_VEL
LIN {X 0,Y 324.026,Z 462.757,A -85,B 0,C 180,E1 -15988.831,E2 -15988.831} C_VEL
LIN {X 0,Y 328.023,Z 468.434,A -85,B 0,C 180,E1 -15990.325,E2 -15990.325} C_VEL
LIN {X 0,Y 331.918,Z 474.923,A -85,B 0,C 180,E1 -15991.665,E2 -15991.665} C_VEL
LIN {X 0,Y 332.662,Z 476.549,A -85,B 0,C 180,E1 -15991.922,E2 -15991.922} C_VEL
LIN {X 0,Y 326.935,Z 533.643,A -85,B 0,C 180,E1 -15994.152,E2 -15994.152} C_VEL
LIN {X 0,Y 325.741,Z 547.254,A -85,B 0,C 180,E1 -15994.822,E2 -15994.822} C_VEL
LIN {X 0,Y 324.198,Z 560.88,A -85,B 0,C 180,E1 -15995.78,E2 -15995.78} C_VEL
LIN {X 0,Y 322.106,Z 574.627,A -85,B 0,C 180,E1 -15997.045,E2 -15997.045} C_VEL
LIN {X 0,Y 319.938,Z 586.112,A -85,B 0,C 180,E1 -15998.411,E2 -15998.411} C_VEL
LIN {X 0,Y 317.672,Z 596.441,A -85,B 0,C 180,E1 -15999.945,E2 -15999.945} C_VEL
LIN {X 0,Y 315.295,Z 606.391,A -85,B 0,C 180,E1 -16001.816,E2 -16001.816} C_VEL
LIN {X 0,Y 313.134,Z 614.423,A -85,B 0,C 180,E1 -16003.707,E2 -16003.707} C_VEL
LIN {X 0,Y 311.222,Z 620.806,A -85,B 0,C 180,E1 -16005.617,E2 -16005.617} C_VEL
LIN {X 0,Y 309.724,Z 625.45,A -85,B 0,C 180,E1 -16007.35,E2 -16007.35} C_VEL
LIN {X 0,Y 308.115,Z 629.844,A -85,B 0,C 180,E1 -16009.486,E2 -16009.486} C_VEL
LIN {X 0,Y 307.254,Z 631.881,A -85,B 0,C 180,E1 -16010.786,E2 -16010.786} C_VEL
LIN {X 0,Y 306.586,Z 633.413,A -85,B 0,C 180,E1 -16012.094,E2 -16012.094} C_VEL
LIN {X 0,Y 306.046,Z 634.493,A -85,B 0,C 180,E1 -16013.407,E2 -16013.407} C_VEL
LIN {X 0,Y 305.541,Z 635.185,A -85,B 0,C 180,E1 -16014.721,E2 -16014.721} C_VEL
LIN {X 0,Y 305.081,Z 635.457,A -85,B 0,C 180,E1 -16016.037,E2 -16016.037} C_VEL
LIN {X 0,Y 304.737,Z 635.259,A -85,B 0,C 180,E1 -16017.356,E2 -16017.356} C_VEL
LIN {X 0,Y 304.523,Z 634.641,A -85,B 0,C 180,E1 -16018.678,E2 -16018.678} C_VEL
LIN {X 0,Y 304.365,Z 633.613,A -85,B 0,C 180,E1 -16020,E2 -16020} C_VEL
LIN {X 0,Y 304.36,Z 632.111,A -85,B 0,C 180,E1 -16021.323,E2 -16021.323} C_VEL
LIN {X 0,Y 304.5,Z 629.04,A -85,B 0,C 180,E1 -16023.308,E2 -16023.308} C_VEL
LIN {X 0,Y 304.666,Z 624.88,A -85,B 0,C 180,E1 -16025.294,E2 -16025.294} C_VEL
LIN {X 0,Y 304.925,Z 618.539,A -85,B 0,C 180,E1 -16027.6,E2 -16027.6} C_VEL
LIN {X 0,Y 305.338,Z 611.49,A -85,B 0,C 180,E1 -16029.606,E2 -16029.606} C_VEL
LIN {X 0,Y 306.029,Z 602.787,A -85,B 0,C 180,E1 -16031.592,E2 -16031.592} C_VEL
LIN {X 0,Y 306.779,Z 592.957,A -85,B 0,C 180,E1 -16033.412,E2 -16033.412} C_VEL
LIN {X 0,Y 307.618,Z 581.887,A -85,B 0,C 180,E1 -16035.063,E2 -16035.063} C_VEL
LIN {X 0,Y 308.456,Z 570.287,A -85,B 0,C 180,E1 -16036.458,E2 -16036.458} C_VEL
LIN {X 0,Y 309.164,Z 557.166,A -85,B 0,C 180,E1 -16037.701,E2 -16037.701} C_VEL
LIN {X 0,Y 309.747,Z 544.677,A -85,B 0,C 180,E1 -16038.607,E2 -16038.607} C_VEL
LIN {X 0,Y 310.289,Z 530.46,A -85,B 0,C 180,E1 -16039.345,E2 -16039.345} C_VEL
LIN {X 0,Y 312.502,Z 457.589,A -85,B 0,C 180,E1 -16041.766,E2 -16041.766} C_VEL
LIN {X 0,Y 305.482,Z 435.426,A -85,B 0,C 180,E1 -16042.865,E2 -16042.865} C_VEL
LIN {X 0,Y 305.528,Z 435.425,A -85,B 0,C 180,E1 -16046.219,E2 -16046.219} C_VEL
LIN {X 0,Y 305.49,Z 435.429,A -85,B 0,C 180,E1 -16049.047,E2 -16049.047} C_VEL
LIN {X 0,Y 305.444,Z 435.426,A -85,B 0,C 180,E1 -16051.952,E2 -16051.952} C_VEL
LIN {X 0,Y 305.464,Z 435.417,A -85,B 0,C 180,E1 -16055.113,E2 -16055.113} C_VEL
LIN {X 0,Y 305.469,Z 435.432,A -85,B 0,C 180,E1 -16058.533,E2 -16058.533} C_VEL
LIN {X 0,Y 305.457,Z 435.437,A -85,B 0,C 180,E1 -16062.586,E2 -16062.586} C_VEL
LIN {X 0,Y 305.427,Z 435.425,A -85,B 0,C 180,E1 -16066.345,E2 -16066.345} C_VEL
LIN {X 0,Y 305.46,Z 435.425,A -85,B 0,C 180,E1 -16069.892,E2 -16069.892} C_VEL
LIN {X 0,Y 305.486,Z 435.426,A -85,B 0,C 180,E1 -16073.631,E2 -16073.631} C_VEL
LIN {X 0,Y 305.475,Z 435.474,A -85,B 0,C 180,E1 -16075.225,E2 -16075.225} C_VEL
LIN {X 0,Y 308.956,Z 448.186,A -85,B 0,C 180,E1 -16078.453,E2 -16078.453} C_VEL
LIN {X 0,Y 311.632,Z 459.906,A -85,B 0,C 180,E1 -16081.237,E2 -16081.237} C_VEL
LIN {X 0,Y 312.842,Z 465.88,A -85,B 0,C 180,E1 -16082.578,E2 -16082.578} C_VEL
LIN {X 0,Y 312.427,Z 473.532,A -85,B 0,C 180,E1 -16084.052,E2 -16084.052} C_VEL
LIN {X 0,Y 317.215,Z 499.911,A -85,B 0,C 180,E1 -16085.138,E2 -16085.138} C_VEL
LIN {X 0,Y 318.021,Z 505.958,A -85,B 0,C 180,E1 -16085.354,E2 -16085.354} C_VEL
LIN {X 0,Y 316.279,Z 580.246,A -85,B 0,C 180,E1 -16087.03,E2 -16087.03} C_VEL
LIN {X 0,Y 315.719,Z 592.942,A -85,B 0,C 180,E1 -16087.462,E2 -16087.462} C_VEL
LIN {X 0,Y 314.741,Z 606.562,A -85,B 0,C 180,E1 -16088.209,E2 -16088.209} C_VEL
LIN {X 0,Y 313.515,Z 618.822,A -85,B 0,C 180,E1 -16089.153,E2 -16089.153} C_VEL
LIN {X 0,Y 312.09,Z 631.12,A -85,B 0,C 180,E1 -16090.429,E2 -16090.429} C_VEL
LIN {X 0,Y 310.68,Z 641.664,A -85,B 0,C 180,E1 -16091.823,E2 -16091.823} C_VEL
LIN {X 0,Y 309.55,Z 649.921,A -85,B 0,C 180,E1 -16093.173,E2 -16093.173} C_VEL
LIN {X 0,Y 307.827,Z 659.613,A -85,B 0,C 180,E1 -16095.117,E2 -16095.117} C_VEL
LIN {X 0,Y 306.598,Z 667.394,A -85,B 0,C 180,E1 -16097.086,E2 -16097.086} C_VEL
LIN {X 0,Y 305.72,Z 672.65,A -85,B 0,C 180,E1 -16098.732,E2 -16098.732} C_VEL
LIN {X 0,Y 304.843,Z 677.787,A -85,B 0,C 180,E1 -16100.713,E2 -16100.713} C_VEL
LIN {X 0,Y 304.342,Z 681.759,A -85,B 0,C 180,E1 -16102.703,E2 -16102.703} C_VEL
LIN {X 0,Y 303.977,Z 684.688,A -85,B 0,C 180,E1 -16104.694,E2 -16104.694} C_VEL
LIN {X 0,Y 303.849,Z 686.107,A -85,B 0,C 180,E1 -16106.021,E2 -16106.021} C_VEL
LIN {X 0,Y 303.611,Z 687.717,A -85,B 0,C 180,E1 -16108.674,E2 -16108.674} C_VEL
LIN {X 0,Y 303.596,Z 687.95,A -85,B 0,C 180,E1 -16110,E2 -16110} C_VEL
LIN {X 0,Y 303.611,Z 687.756,A -85,B 0,C 180,E1 -16111.326,E2 -16111.326} C_VEL
LIN {X 0,Y 303.848,Z 686.197,A -85,B 0,C 180,E1 -16113.979,E2 -16113.979} C_VEL
LIN {X 0,Y 303.976,Z 684.829,A -85,B 0,C 180,E1 -16115.306,E2 -16115.306} C_VEL
LIN {X 0,Y 304.335,Z 681.953,A -85,B 0,C 180,E1 -16117.297,E2 -16117.297} C_VEL
LIN {X 0,Y 304.839,Z 678.044,A -85,B 0,C 180,E1 -16119.287,E2 -16119.287} C_VEL
LIN {X 0,Y 305.654,Z 672.975,A -85,B 0,C 180,E1 -16121.271,E2 -16121.271} C_VEL
LIN {X 0,Y 306.721,Z 666.583,A -85,B 0,C 180,E1 -16123.246,E2 -16123.246} C_VEL
LIN {X 0,Y 308.087,Z 658.639,A -85,B 0,C 180,E1 -16125.209,E2 -16125.209} C_VEL
LIN {X 0,Y 309.467,Z 650.514,A -85,B 0,C 180,E1 -16126.831,E2 -16126.831} C_VEL
LIN {X 0,Y 310.844,Z 640.518,A -85,B 0,C 180,E1 -16128.453,E2 -16128.453} C_VEL
